(* IEC 61131-3 sources: volt/packages/volt-lsp-iec/test-corpus/lenze-mid/Device/Plc Logic/Application/A70_MachineModuleSources/MM_MachineControl/01_Main, 9 files *)

(* ---- Mach1_Drives.pou ---- *)
FUNCTION_BLOCK Mach1_Drives
VAR_INPUT
END_VAR
VAR_OUTPUT
END_VAR
VAR
	testbyte: BYTE;
	testdint: DWORD;
	testword: WORD;
	OspRotationFlag: R_TRIG;
	OffDelayEnableDrivePower: TOF;
	EnableDrivePower: BOOL;
	bServoDrivesInSync: BOOL;
	TimeOutInSync: TON;
	bInSyncTimeOut: BOOL;
	TimeOutInLock: TON;
	tSetDrivesInLock: BOOL;
	bInLockTimeOut: BOOL;
	SideCorrection_CW: sUDT_ServoComm_Drive_Control;
	Servo_LimitJog_Instance: Servo_LimitJog;
	FBFeedforwardADS: FB_Lenze_i550;
	FBFeedforwardATF: FB_Lenze_i550;
	FBElevatorATF: FB_Lenze_i550;
	FBFan: FB_Lenze_i550;
	FBBobbin: FB_Lenze_i550;
	tReal: REAL;
	tWrapperStopPosition: DINT;

	sadad: FB_Lenze_i550;
	FB_Lenze_i550_0: FB_Lenze_i550;

mydword:DWORD;

	tbool: BOOL;
	OnDelayEnableSync: TON;
	ScaleBobbinTorque: LIN_TRAFO;
	tBobbinTorque: REAL;
	OffDelaySync: TOF;
	TON_0: TON;

	MainDrive_VirtualMasterControl: VirtualMasterControl;
END_VAR

VAR CONSTANT
	ctCurveIsSpeed: INT := 2;
	ctCurveIs0ToMax: INT := 0;
END_VAR
VAR
	ServoMainDrive: ServoControl;
	ServoWrappingDevice: ServoControl;
	ServoSideCorrection: ServoControl;
END_VAR
%LANGUAGE LD
%NETWORK "DONE network 3 : All drives ready"
ASSIGN((Mach1_Data.Drives.MainDrive.Status.DriveIsReady OR INVERT(Mach1_Data.Drives.MainDrive.Control.SetDriveEnable)) AND (Mach1_Data.Drives.WrappingDevice.Status.DriveIsReady OR INVERT(Mach1_Data.Drives.WrappingDevice.Control.SetDriveEnable)) AND (Mach1_Data.Drives.SideCorrection.Status.DriveIsReady OR INVERT(Mach1_Data.Drives.SideCorrection.Control.SetDriveEnable)), Q => Mach1.GenFlags.ConditionsReadyForOperation);
%NETWORK
VAR w1 : ANY; END_VAR
w1 := EnableDrivePower;
ASSIGN(w1 AND Mach1_Data.Drives.WrappingDevice.Status.DriveIsHomed, Q_RESET => Mach1_Data.Drives.WrappingDevice.Control.StartSetHomePos);
ASSIGN((w1 AND INVERT(Mach1_Data.Drives.WrappingDevice.Status.DriveIsHomed)) AND FF500ms, Q_SET => Mach1_Data.Drives.WrappingDevice.Control.StartSetHomePos);
%NETWORK "DONE Network 4: Enable drive power "
// The off delay ensures that the drive can stop before the power is removed from the drive. The power must be removed from the drive before it goes to STO. If the power remains on during STO, the drive will generate an error.
ASSIGN(TRUE AND Mach1_Safety.Status.STO_OK, Q => EnableDrivePower);
%NETWORK
ASSIGN(Mach1_Data.Drives.MainDrive.Status.DriveIsHomed, Q => Mach1_AuxData.AllDrivesHomed);
%NETWORK
VAR w2 : ANY; END_VAR
w2 := TRUE;
ASSIGN(w2 AND mach1.Genflags.DelayAfterSTO, Q => Mach1_Data.Drives.MainDrive_VM.Control.SetDriveEnable);
ASSIGN((w2 AND INVERT(Mach1_Data.Drives.MainDrive_VM.Status.DriveIsReady)) AND FF100ms, Q => Mach1_Data.Drives.MainDrive_VM.Control.ResetError);
MainDrive_VirtualMasterControl(EN := w2, iAcc := 600, iDec := 1800, ioVirtualMaster := Mach1_Data.Drives.MainDrive_VM, ioVirtualMasterCom := Data_Exchange_Motion.Servo_VirtualMaster);
MOVE(EN := MOVE(EN := w2, Mach1_Data.Drives.MainDrive_VM.Status.ActSpeed, OUT => HMI_Var.Mach1.ActualSpeed), Mach1_Data.Drives.MainDrive_VM.Status.ActXPos, OUT => HMI_Var.Mach1.Position);
%NETWORK "Warning: machine in manual homing mode"
Alarms_V5_1_100(AlarmDB := Mach1_Alarms, iCond := Mach1.GenFlags.DelayAfterSTO AND Mach1_AuxData.EnableManualHomeSetting, iReset := Mach1.GenFlags.ResetFlag, iAlm := Mach1_Alarms.Alm033, ioAction := Mach1.GenFlags.Warning);
%NETWORK "DONE Network 5 : Conditions for sync/lock"
VAR w3 : ANY; w4 : ANY; w5 : ANY; END_VAR
w3 := Mach1.GenFlags.DelayAfterEmergStop;
ASSIGN(TON_0(IN := OffDelaySync(IN := w3 AND Mach1_Safety.Status.DoorsOK, PT := T#500MS) AND Mach1_Safety.Status.STO_OK, PT := T#500MS) AND Mach1.GenFlags.ConditionsReadyForOperation AND Mach1_AuxData.AllDrivesHomed AND INVERT(Mach1_AuxData.EnableManualHomeSetting), Q => Mach1_AuxData.SetDrivesInSync);
w4 := w3 AND Mach1_AuxData.SetDrivesInSync;
ASSIGN(w4 AND Mach1_Data.Drives.MainDrive.Status.InSync AND (Mach1_Data.Drives.WrappingDevice.Status.InSync OR INVERT(Mach1_Data.Drives.WrappingDevice.Control.SetDriveEnable)) AND (Mach1_Data.Drives.SideCorrection.Status.InSync OR INVERT(Mach1_Data.Drives.SideCorrection.Control.SetDriveEnable)), Q => bServoDrivesInSync);
ASSIGN(TimeOutInSync(IN := w4 AND INVERT(bServoDrivesInSync), PT := T#10S), Q => bInSyncTimeOut);
ASSIGN(BRANCH_SHORTCIRCUIT(FEED := w3 AND bServoDrivesInSync, Mach1_AuxData.IEC_TIMERS.OffDelayLockDrives(IN := RAIL(), PT := T#2s), TRUE), Q => Mach1_AuxData.SetDrivesInLock);
w5 := w3 AND (Mach1_AuxData.SetDrivesInLock OR Mach1_AuxData.SetDrivesInSync);
ASSIGN(w5 AND Mach1_Data.Drives.MainDrive.Status.InSync AND (Mach1_Data.Drives.WrappingDevice.Status.InSync OR INVERT(Mach1_Data.Drives.WrappingDevice.Control.SetDriveEnable)) AND (Mach1_Data.Drives.SideCorrection.Status.InSync OR INVERT(Mach1_Data.Drives.SideCorrection.Control.SetDriveEnable)), Q => Mach1_AuxData.AllDrivesInLock);
ASSIGN(TimeOutInLock(IN := w5 AND INVERT(Mach1_AuxData.AllDrivesInLock), PT := T#5S), Q => bInLockTimeOut);
ASSIGN(w5, Q => tSetDrivesInLock);
%NETWORK "DONE Network 6: Servo Main drive: Control"
VAR w6 : ANY; w7 : ANY; END_VAR
w6 := TRUE;
ASSIGN(w6 AND (Mach1_Safety.Control.RequestManSpeed AND Mach1_Safety.Status.SafetyManSpeed OR Mach1_Safety.Control.RequestAutoSpeed AND Mach1_Safety.Status.SafetyAutoSpeed), Q => Mach1_Data.Drives.MainDrive_VM.Control.StartMovement);
ASSIGN(MOVE(EN := w6 AND TRUE, ctCurveIs0ToMax, OUT => Mach1_Data.Drives.MainDrive.CAM.CamType) AND tSetDrivesInLock, Q => Mach1_Data.Drives.MainDrive.Control.SetInSync);
w7 := w6 AND TRUE;
ASSIGN(w7 AND Mach1_Alarms.Alm001 AND HMI_Var.ReleaseBrake, Q => Mach1_Data.Drives.MainDrive.Control.SetBrakeRelease);
ASSIGN(w7 AND (INVERT(Mach1_Alarms.Alm001) OR mach1.Genflags.StartFlag AND Mach1_Alarms.Alm001), Q_RESET => HMI_Var.ReleaseBrake);
ASSIGN(OspRotationFlag(CLK := ServoMainDrive(EN := w6 AND TRUE, iServoStatus := Data_Exchange_Motion.Servo_MainDrive.Status, iEnableHomeMovement := TRUE, iEnablePower := EnableDrivePower, iFF100ms := LST_General.FF100ms, ioUDT_ServoDrive := Mach1_Data.Drives.MainDrive, oServoControl => Data_Exchange_Motion.Servo_MainDrive.Control) AND Mach1_Data.Drives.MainDrive.Status.RotationPulse), Q => Mach1.GenFlags.Rotflag);
%NETWORK "DONE Network 7 : Servo Main drive: Alarms"
ASSIGN(Alarms_V5_1_100(AlarmDB := Mach1_Alarms, iCond := Mach1.GenFlags.DelayAfterSTO AND INVERT(Mach1_Data.Drives.MainDrive.Status.DriveIsReady), iReset := Mach1.GenFlags.ResetFlag, iAlm := Mach1_Alarms.Alm020, ioAction := Mach1.GenFlags.MinorAlarm) OR Alarms_V5_1_100(AlarmDB := Mach1_Alarms, iCond := Mach1.GenFlags.DelayAfterSTO AND Mach1_Data.Drives.MainDrive.Status.DriveTorqueError, iReset := Mach1.GenFlags.ResetFlag, iAlm := Mach1_Alarms.Alm021, ioAction := Mach1.GenFlags.MinorAlarm) OR Alarms_V5_1_100(AlarmDB := Mach1_Alarms, iCond := Mach1.GenFlags.DelayAfterSTO AND INVERT(Mach1_Data.Drives.MainDrive.Status.DriveIsHomed), iReset := Mach1.GenFlags.ResetFlag, iAlm := Mach1_Alarms.Alm022, ioAction := Mach1.GenFlags.MinorAlarm), Q_SET => Mach1.GenFlags.StopDriveDirect);
%NETWORK
ASSIGN((Mach1_Alarms.Alm020 OR Mach1_Alarms.Alm021 OR Mach1_Alarms.Alm022) AND Mach1.GenFlags.ResetFlag OR TON_0.Q AND Imp100ms AND Mach1_Safety.Status.ServiceMode AND Mach1_Safety.Status.Service_ButtonAB, Q_SET => Mach1_Data.Drives.MainDrive.Control.ResetError);
%NETWORK "DONE Network 8: Servo Wrapping device: Control"
VAR w8 : ANY; END_VAR
w8 := TRUE;
ASSIGN(MOVE(EN := w8 AND TRUE, ctCurveIsSpeed, OUT => Mach1_Data.Drives.WrappingDevice.CAM.CamType) AND tSetDrivesInLock, Q => Mach1_Data.Drives.WrappingDevice.Control.SetInSync);
MOVE(EN := w8, Mach1_Data.Settings.Ints.RollingDeviceSpeedFactor, OUT => Mach1_Data.Drives.WrappingDevice.CAM.Y_Scale_Recipe);
ServoWrappingDevice(EN := w8 AND TRUE, iServoStatus := Data_Exchange_Motion.Servo_WrappingDevice.Status, iEnableHomeMovement := TRUE, iEnablePower := EnableDrivePower, iFF100ms := LST_General.FF100ms, ioUDT_ServoDrive := Mach1_Data.Drives.WrappingDevice, oServoControl => Data_Exchange_Motion.Servo_WrappingDevice.Control);
%NETWORK "DONE Network 9 : Servo Wrapping Device: Alarms"
VAR w9 : ANY; END_VAR
w9 := Alarms_V5_1_100(AlarmDB := Mach1_Alarms, iCond := Mach1.GenFlags.DelayAfterSTO AND INVERT(Mach1_Data.Drives.WrappingDevice.Status.DriveIsReady) AND Mach1_Data.Drives.WrappingDevice.Control.SetDriveEnable, iReset := Mach1.GenFlags.ResetFlag, iAlm := Mach1_Alarms.Alm023, ioAction := Mach1.GenFlags.MinorAlarm) OR Alarms_V5_1_100(AlarmDB := Mach1_Alarms, iCond := Mach1.GenFlags.DelayAfterSTO AND Mach1_Data.Drives.WrappingDevice.Status.DriveTorqueError, iReset := Mach1.GenFlags.ResetFlag, iAlm := Mach1_Alarms.Alm024, ioAction := Mach1.GenFlags.MinorAlarm) OR Alarms_V5_1_100(AlarmDB := Mach1_Alarms, iCond := Mach1.GenFlags.DelayAfterSTO AND INVERT(Mach1_Data.Drives.WrappingDevice.Status.DriveIsHomed), iReset := Mach1.GenFlags.ResetFlag, iAlm := Mach1_Alarms.Alm025, ioAction := Mach1.GenFlags.MinorAlarm);
ASSIGN(w9, Q_SET => Mach1.GenFlags.StopDriveDirect);
ASSIGN(w9 AND Mach1.GenFlags.ResetFlag, Q_SET => Mach1_Data.Drives.WrappingDevice.Control.ResetError);
%NETWORK
ASSIGN((Mach1_Alarms.Alm023 OR Mach1_Alarms.Alm024 OR Mach1_Alarms.Alm025) AND Mach1.GenFlags.ResetFlag OR TON_0.Q AND Imp100ms AND Mach1_Safety.Status.ServiceMode AND Mach1_Safety.Status.Service_ButtonAB, Q_SET => Mach1_Data.Drives.WrappingDevice.Control.ResetError);
%NETWORK
%NETWORK "Digital inputs"
VAR w10 : ANY; END_VAR
// 16: non-motor side
// 17: motor side
w10 := MOVE(EN := TRUE, %ID79, OUT => mydword);
ASSIGN(w10 AND mydword.16, Q => Data_Exchange_Motion.Servo_SideCorrection.Status.Spare1);
ASSIGN(w10 AND mydword.17, Q => Data_Exchange_Motion.Servo_SideCorrection.Status.Spare2);
%NETWORK "DONE Network 10: Servo Side correction: Control"
VAR w11 : ANY; END_VAR
w11 := TRUE;
ASSIGN(MOVE(EN := w11 AND TRUE, ctCurveIsSpeed, OUT => Mach1_Data.Drives.SideCorrection.CAM.CamType) AND tSetDrivesInLock, Q => Mach1_Data.Drives.SideCorrection.Control.SetInSync);
ServoSideCorrection(EN := w11 AND TRUE, iServoStatus := Data_Exchange_Motion.Servo_SideCorrection.Status, iEnableHomeMovement := TRUE, iEnablePower := EnableDrivePower, iFF100ms := LST_General.FF100ms, ioUDT_ServoDrive := Mach1_Data.Drives.SideCorrection, oServoControl => SideCorrection_CW);
Servo_LimitJog_Instance(EN := w11 AND TRUE, iServoStatus := Data_Exchange_Motion.Servo_SideCorrection.Status, iServoControl := SideCorrection_CW, ioUDT_ServoDrive := Mach1_Data.Drives.SideCorrection, ioUDT_JogLimitFree := Mach1_Data.Drives.SideCorrection_FreeLimit, oServoControl => Data_Exchange_Motion.Servo_SideCorrection.Control);
%NETWORK "DONE Network 11 : Servo Side correction: Alarms"
VAR w12 : ANY; END_VAR
w12 := Alarms_V5_1_100(AlarmDB := Mach1_Alarms, iCond := Mach1.GenFlags.DelayAfterSTO AND INVERT(Mach1_Data.Drives.SideCorrection.Status.DriveIsReady) AND Mach1_Data.Drives.SideCorrection.Control.SetDriveEnable, iReset := Mach1.GenFlags.ResetFlag, iAlm := Mach1_Alarms.Alm026, ioAction := Mach1.GenFlags.MinorAlarm) OR Alarms_V5_1_100(AlarmDB := Mach1_Alarms, iCond := Mach1.GenFlags.DelayAfterSTO AND Mach1_Data.Drives.SideCorrection.Status.DriveTorqueError, iReset := Mach1.GenFlags.ResetFlag, iAlm := Mach1_Alarms.Alm027, ioAction := Mach1.GenFlags.MinorAlarm) OR Alarms_V5_1_100(AlarmDB := Mach1_Alarms, iCond := Mach1.GenFlags.DelayAfterSTO AND INVERT(Mach1_Data.Drives.SideCorrection.Status.DriveIsHomed), iReset := Mach1.GenFlags.ResetFlag, iAlm := Mach1_Alarms.Alm028, ioAction := Mach1.GenFlags.MinorAlarm);
ASSIGN(w12, Q_SET => Mach1.GenFlags.StopDriveDirect);
ASSIGN(w12 AND Mach1.GenFlags.ResetFlag, Q_SET => Mach1_Data.Drives.SideCorrection.Control.ResetError);
%NETWORK
ASSIGN((Mach1_Alarms.Alm026 OR Mach1_Alarms.Alm027 OR Mach1_Alarms.Alm028) AND Mach1.GenFlags.ResetFlag OR TON_0.Q AND Imp100ms AND Mach1_Safety.Status.ServiceMode AND Mach1_Safety.Status.Service_ButtonAB, Q_SET => Mach1_Data.Drives.SideCorrection.Control.ResetError);
%NETWORK
%NETWORK "DONE Network 12: Feedforward ADS"
VAR w13 : ANY; END_VAR
w13 := TRUE;
ASSIGN(w13 AND Mach1.GenFlags.DelayAfterEmergStop AND INVERT(Mach1_Alarms.Alm015), Q => Mach1_Data.Drives.FeedForwardADS.Control.Enable);
ASSIGN(w13, Q => Mach1_Data.Drives.FeedForwardADS.Control.Reverse);
FBFeedforwardADS(EN := w13, iStatusWord := Data_Exchange_Motion.FQI_FeedforwardADS.Status, iGearRatioNumerator := 2790.0, iGearRatioDenominator := 111.0, iNominalMotorSpeedwoSlipComp_RPM := 3000.0, iNominalMotorFrequency_Hz := 100.0, iAxisJogSpeed_RPM := 10.0, ioUDT := Mach1_Data.Drives.FeedForwardADS, oControlWord => Data_Exchange_Motion.FQI_FeedforwardADS.Controlword, oRefSpeed => Data_Exchange_Motion.FQI_FeedforwardADS.RefSpeed);
%NETWORK "DONE Network 13: Alarms feed forward dryer "
VAR w14 : ANY; END_VAR
w14 := Alarms_V5_1_100(AlarmDB := Mach1_Alarms, iCond := Mach1.GenFlags.DelayAfterEmergStop AND Mach1_Data.Drives.FeedForwardADS.Status.Error, iReset := True, iAlm := Mach1_Alarms.Alm015, ioAction := Mach1.GenFlags.MinorAlarm);
ASSIGN(w14, Q_SET => Mach1.GenFlags.StopDriveDirect);
ASSIGN(w14 AND Mach1.GenFlags.ResetFlag, Q_SET => Mach1_Data.Drives.FeedForwardADS.Control.ResetError);
%NETWORK "DONE Network 14: Feedforward ATF"
VAR w15 : ANY; END_VAR
w15 := TRUE;
ASSIGN(w15 AND Mach1.GenFlags.DelayAfterEmergStop AND INVERT(Mach1_Alarms.Alm016), Q => Mach1_Data.Drives.FeedForwardATF.Control.Enable);
FBFeedforwardATF(EN := w15, iStatusWord := Data_Exchange_Motion.FQI_FeedforwardATF.Status, iGearRatioNumerator := 2790.0, iGearRatioDenominator := 111.0, iNominalMotorSpeedwoSlipComp_RPM := 3000.0, iNominalMotorFrequency_Hz := 100.0, iAxisJogSpeed_RPM := 10.0, ioUDT := Mach1_Data.Drives.FeedForwardATF, oControlWord => Data_Exchange_Motion.FQI_FeedforwardATF.Controlword, oRefSpeed => Data_Exchange_Motion.FQI_FeedforwardATF.RefSpeed);
%NETWORK "DONE Network 15: Alarms feed forward trayfiller$R$L"
VAR w16 : ANY; END_VAR
w16 := Alarms_V5_1_100(AlarmDB := Mach1_Alarms, iCond := Mach1.GenFlags.DelayAfterEmergStop AND Mach1_Data.Drives.FeedForwardATF.Status.Error, iReset := True, iAlm := Mach1_Alarms.Alm016, ioAction := Mach1.GenFlags.MinorAlarm);
ASSIGN(w16, Q_SET => Mach1.GenFlags.StopDriveDirect);
ASSIGN(w16 AND Mach1.GenFlags.ResetFlag, Q_SET => Mach1_Data.Drives.FeedForwardATF.Control.ResetError);
%NETWORK "DONE Network 16: Elevator ATF"
VAR w17 : ANY; END_VAR
w17 := TRUE;
ASSIGN(w17 AND Mach1.GenFlags.DelayAfterEmergStop AND INVERT(Mach1_Alarms.Alm014), Q => Mach1_Data.Drives.ElevatorATF.Control.Enable);
FBElevatorATF(EN := w17, iStatusWord := Data_Exchange_Motion.FQI_ElevatorATF.Status, iGearRatioNumerator := 100.0, iGearRatioDenominator := 111.0, iNominalMotorSpeedwoSlipComp_RPM := 3000.0, iNominalMotorFrequency_Hz := 100.0, iAxisJogSpeed_RPM := 10.0, ioUDT := Mach1_Data.Drives.ElevatorATF, oControlWord => Data_Exchange_Motion.FQI_ElevatorATF.Controlword, oRefSpeed => Data_Exchange_Motion.FQI_ElevatorATF.RefSpeed);
%NETWORK "DONE Network 17: Alarms Elevator trayfiller$R$L"
VAR w18 : ANY; END_VAR
w18 := Alarms_V5_1_100(AlarmDB := Mach1_Alarms, iCond := Mach1.GenFlags.DelayAfterEmergStop AND Mach1_Data.Drives.ElevatorATF.Status.Error, iReset := True, iAlm := Mach1_Alarms.Alm014, ioAction := Mach1.GenFlags.MinorAlarm);
ASSIGN(w18, Q_SET => Mach1.GenFlags.StopDriveDirect);
ASSIGN(w18 AND Mach1.GenFlags.ResetFlag, Q_SET => Mach1_Data.Drives.ElevatorATF.Control.ResetError);
%NETWORK "DONE Network 18: Fan"
VAR w19 : ANY; END_VAR
w19 := TRUE;
ASSIGN(w19 AND Mach1.GenFlags.EnableAuxDrive AND INVERT(Mach1_Alarms.Alm017), Q => Mach1_Data.Drives.Fan.Control.Enable);
FBFan(EN := w19, iStatusWord := Data_Exchange_Motion.FQI_Fan.Status, iGearRatioNumerator := 1.0, iGearRatioDenominator := 1.0, iNominalMotorSpeedwoSlipComp_RPM := 3000.0, iNominalMotorFrequency_Hz := 50.0, iAxisJogSpeed_RPM := 10.0, ioUDT := Mach1_Data.Drives.Fan, oControlWord => Data_Exchange_Motion.FQI_Fan.Controlword, oRefSpeed => Data_Exchange_Motion.FQI_Fan.RefSpeed);
%NETWORK "DONE Network 19: Alarms Fan$R$L"
VAR w20 : ANY; END_VAR
w20 := Alarms_V5_1_100(AlarmDB := Mach1_Alarms, iCond := Mach1.GenFlags.DelayAfterEmergStop AND Mach1_Data.Drives.Fan.Status.Error, iReset := True, iAlm := Mach1_Alarms.Alm017, ioAction := Mach1.GenFlags.MinorAlarm);
ASSIGN(w20, Q_SET => Mach1.GenFlags.StopDriveDirect);
ASSIGN(w20 AND Mach1.GenFlags.ResetFlag, Q_SET => Mach1_Data.Drives.Fan.Control.ResetError);
%NETWORK "DONE Network 20: Bobbin"
VAR w21 : ANY; w22 : ANY; w23 : ANY; END_VAR
w21 := TRUE;
w22 := GT(EN := w21 AND Mach1.GenFlags.EnableAuxDrive AND INVERT(HMI_Var.Btn_Cleaning), Mach1_Data.Settings.Ints.TorqueControlBobbin, 0).OUT AND Mach1_Safety.Status.AllDoorsActuallyClosed;
ASSIGN(w22, Q => Mach1_Data.Drives.Bobbine.Control.Enable);
ASSIGN(MOVE(EN := w22, 860, OUT => Mach1_Data.Drives.Bobbine.Control.AutoSpeed), Q => Mach1_Data.Drives.Bobbine.Control.StartAuto);
FBBobbin(EN := w21, iStatusWord := Data_Exchange_Motion.FQI_Bobbin.Status, iGearRatioNumerator := 2790.0, iGearRatioDenominator := 111.0, iNominalMotorSpeedwoSlipComp_RPM := 3000.0, iNominalMotorFrequency_Hz := 50.0, iAxisJogSpeed_RPM := 10.0, ioUDT := Mach1_Data.Drives.Bobbine, oControlWord => Data_Exchange_Motion.FQI_Bobbin.Controlword, oRefSpeed => Data_Exchange_Motion.FQI_Bobbin.RefSpeed);
w23 := w21 AND HMI_Var.Mach1.CalibrateTorqueValues;
MOVE(EN := w23, Mach1_AuxData.TorqueCalibrationValue, OUT => Data_Exchange_Motion.BobbinTorque);
ASSIGN(MOVE(EN := w23 AND HMI_Var.Mach1.setMinTorqueValue, Mach1_AuxData.TorqueCalibrationValue, OUT => Mach1_Data.Settings.Dints.minTorqueValue), Q_RESET => HMI_Var.Mach1.setMinTorqueValue);
ASSIGN(MOVE(EN := w23 AND HMI_Var.Mach1.setMaxTorqueValue, Mach1_AuxData.TorqueCalibrationValue, OUT => Mach1_Data.Settings.Dints.maxTorqueValue), Q_RESET => HMI_Var.Mach1.setMaxTorqueValue);
MOVE(EN := ScaleBobbinTorque(EN := w21 AND INVERT(HMI_Var.Mach1.CalibrateTorqueValues), IN := Mach1_Data.Settings.Ints.TorqueControlBobbin, IN_MIN := 0, IN_MAX := 1000, OUT_MIN := OPERAND('DINT_TO_REAL(Mach1_Data.Settings.Dints.minTorqueValue)'), OUT_MAX := OPERAND('DINT_TO_REAL(Mach1_Data.Settings.Dints.maxTorqueValue)'), OUT => tBobbinTorque), OPERAND('REAL_TO_DINT(tBobbinTorque)'), OUT => Data_Exchange_Motion.BobbinTorque);
%NETWORK "DONE Network 21: Alarms Bobbine $R$L"
VAR w24 : ANY; END_VAR
w24 := Alarms_V5_1_100(AlarmDB := Mach1_Alarms, iCond := Mach1_AuxData.MIDS_Active AND Mach1.GenFlags.DelayAfterEmergStop AND INVERT(Mach1_Data.Drives.Bobbine.Status.DriveReady) AND Mach1_AuxData.AllDrivesHomed, iReset := True, iAlm := Mach1_Alarms.Alm010, ioAction := Mach1.GenFlags.MinorAlarm);
ASSIGN(w24, Q_SET => Mach1.GenFlags.StopDriveDirect);
ASSIGN(w24 AND Mach1.GenFlags.ResetFlag, Q_SET => Mach1_Data.Drives.Bobbine.Control.ResetError);
%NETWORK "TODO Network 22:"
// WRAPPER
%NETWORK "TODO Network 23: Limit Wrapper stop position"
VAR w25 : ANY; END_VAR
w25 := TRUE;
MOVE(EN := GT(EN := w25, Mach1_Data.Settings.Dints.WrapperStopPosition, 400).OUT, 400, OUT => Mach1_Data.Settings.Dints.WrapperStopPosition);
MOVE(EN := LT(EN := w25, Mach1_Data.Settings.Dints.WrapperStopPosition, 5).OUT, 5, OUT => Mach1_Data.Settings.Dints.WrapperStopPosition);
MUL(EN := w25, Mach1_Data.Settings.Dints.WrapperStopPosition, 100, OUT => tWrapperStopPosition);
%NETWORK "TODO Network 25:"
ASSIGN(TRUE AND Mach1.GenFlags.DelayAfterEmergStop AND INVERT(Mach1_Alarms.Alm066), Q => Data_Exchange_Motion.FeedForwardWrapper.Control.Enable);
%NETWORK "TODO Network 26:"
ASSIGN(Alarms_V5_1_100(AlarmDB := Mach1_Alarms, iCond := Mach1_AuxData.MIDS_Active AND Mach1.GenFlags.EnableMainDrive AND HMI_Var.Test_Prod AND INVERT(HMI_Var.Btn_Cleaning) AND Mach1_AuxData.AllDrivesHomed AND INVERT(Data_Exchange_Motion.FeedForwardWrapper.Status.ReadyForMotion), iReset := Mach1.Genflags.StartFlag, iAlm := Mach1_Alarms.Alm056, ioAction := Mach1.GenFlags.MinorAlarm) AND mach1.Genflags.ResetFlag, Q_SET => Mach1_Data.Drives.WrappingDevice.Control.ResetError, Q => Data_Exchange_Motion.FeedForwardWrapper.Control.ResetError);
%NETWORK "TODO Network 27:"
;

END_FUNCTION_BLOCK

(* ---- fc_Information.pou ---- *)
PROGRAM fc_Information
VAR
END_VAR

%LANGUAGE ST
VersionInfo_DB.PLC_version:='MID-S100-L-V00_00';
VersionInfo_DB.PLC_Version_Date:='08-06-2023';

END_PROGRAM

(* ---- ForceOutput.pou ---- *)
PROGRAM ForceOutput
VAR
END_VAR

%LANGUAGE LD
%NETWORK
VAR w1 : ANY; END_VAR
w1 := HMI_Var.ForceOutputs;
ASSIGN(w1 AND LST_InputsOutputs.Serv_QB100.0, Q => LST_InputsOutputs.Q100_0_Pilot_light_Alarm_green_);
ASSIGN(w1 AND LST_InputsOutputs.Serv_QB100.1, Q => LST_InputsOutputs.Q100_1_Pilot_light_Alarm_orange_);
ASSIGN(w1 AND LST_InputsOutputs.Serv_QB100.2, Q => LST_InputsOutputs.Q100_2_Pilot_light_Alarm_red_);
ASSIGN(w1 AND LST_InputsOutputs.Serv_QB100.3, Q => LST_InputsOutputs.Q100_3_Pilot_light_Alarm_buzzer_);
ASSIGN(w1 AND LST_InputsOutputs.Serv_QB100.4, Q => LST_InputsOutputs.Q100_4_Spare);
ASSIGN(w1 AND LST_InputsOutputs.Serv_QB100.5, Q => LST_InputsOutputs.Q100_5_Signal_lamp_Start);
ASSIGN(w1 AND LST_InputsOutputs.Serv_QB100.6, Q => LST_InputsOutputs.Q100_6_Signal_lamp_Stop);
ASSIGN(w1 AND LST_InputsOutputs.Serv_QB100.7, Q => LST_InputsOutputs.Q100_7_Activate_greasing_system);
ASSIGN(w1 AND LST_InputsOutputs.Serv_QB101.0, Q => LST_InputsOutputs.Q101_0_REL_release_brake);
ASSIGN(w1 AND LST_InputsOutputs.Serv_QB101.1, Q => LST_InputsOutputs.Q101_1_PNV_Waterlevel_control);
ASSIGN(w1 AND LST_InputsOutputs.Serv_QB101.2, Q => LST_InputsOutputs.Q101_2_Enable_GluePump);
ASSIGN(w1 AND LST_InputsOutputs.Serv_QB101.3, Q => LST_InputsOutputs.Q101_3_Spare);
ASSIGN(w1 AND LST_InputsOutputs.Serv_QB101.4, Q => LST_InputsOutputs.Q101_4_Spare);
ASSIGN(w1 AND LST_InputsOutputs.Serv_QB101.5, Q => LST_InputsOutputs.Q101_5_Spare);
ASSIGN(w1 AND LST_InputsOutputs.Serv_QB101.6, Q => LST_InputsOutputs.Q101_6_Spare);
ASSIGN(w1 AND LST_InputsOutputs.Serv_QB101.7, Q => LST_InputsOutputs.Q101_7_Spare);
%NETWORK
VAR w2 : ANY; END_VAR
w2 := HMI_Var.ForceOutputs;
ASSIGN(w2 AND LST_InputsOutputs.Serv_QB132.0, Q => LST_InputsOutputs.Q132_0_SL_Start_OP2a);
ASSIGN(w2 AND LST_InputsOutputs.Serv_QB132.1, Q => LST_InputsOutputs.Q132_1_SL_Stop_OP2a);
ASSIGN(w2 AND LST_InputsOutputs.Serv_QB132.2, Q => LST_InputsOutputs.Q132_2_Enable_power_controllers);
ASSIGN(w2 AND LST_InputsOutputs.Serv_QB132.3, Q => LST_InputsOutputs.Q132_3_Spare);
ASSIGN(w2 AND LST_InputsOutputs.Serv_QB132.4, Q => LST_InputsOutputs.Q132_4_CT_Fan_dryer);
ASSIGN(w2 AND LST_InputsOutputs.Serv_QB132.5, Q => LST_InputsOutputs.Q132_5_Spare);
ASSIGN(w2 AND LST_InputsOutputs.Serv_QB132.6, Q => LST_InputsOutputs.Q132_6_PNV_Inpusher);
ASSIGN(w2 AND LST_InputsOutputs.Serv_QB132.7, Q => LST_InputsOutputs.Q132_7_PNV_tilting_inpusher);
ASSIGN(w2 AND LST_InputsOutputs.Serv_QB133.0, Q => LST_InputsOutputs.Q133_0_Spare);
ASSIGN(w2 AND LST_InputsOutputs.Serv_QB133.1, Q => LST_InputsOutputs.Q133_1_Spare);
ASSIGN(w2 AND LST_InputsOutputs.Serv_QB133.2, Q => LST_InputsOutputs.Q133_2_Spare);
ASSIGN(w2 AND LST_InputsOutputs.Serv_QB133.3, Q => LST_InputsOutputs.Q133_3_Spare);
ASSIGN(w2 AND LST_InputsOutputs.Serv_QB133.4, Q => LST_InputsOutputs.Q133_4_Spare);
ASSIGN(w2 AND LST_InputsOutputs.Serv_QB133.5, Q => LST_InputsOutputs.Q133_5_InfeedConv_Fwd);
ASSIGN(w2 AND LST_InputsOutputs.Serv_QB133.6, Q => LST_InputsOutputs.Q133_6_InfeedConv_Rev);
ASSIGN(w2 AND LST_InputsOutputs.Serv_QB133.7, Q => LST_InputsOutputs.Q133_7_OutfeedConv_Fwd);
%NETWORK
VAR w3 : ANY; END_VAR
w3 := HMI_Var.ForceOutputs;
ASSIGN(w3 AND LST_InputsOutputs.Serv_QB136.0, Q => LST_InputsOutputs.Q136_0_Spare);
ASSIGN(w3 AND LST_InputsOutputs.Serv_QB136.1, Q => LST_InputsOutputs.Q136_1_Spare);
ASSIGN(w3 AND LST_InputsOutputs.Serv_QB136.2, Q => LST_InputsOutputs.Q136_2_Spare);
ASSIGN(w3 AND LST_InputsOutputs.Serv_QB136.3, Q => LST_InputsOutputs.Q136_3_Spare);
ASSIGN(w3 AND LST_InputsOutputs.Serv_QB136.4, Q => LST_InputsOutputs.Q136_4_Spare);
ASSIGN(w3 AND LST_InputsOutputs.Serv_QB136.5, Q => LST_InputsOutputs.Q136_5_Spare);
ASSIGN(w3 AND LST_InputsOutputs.Serv_QB136.6, Q => LST_InputsOutputs.Q136_6_Spare);
ASSIGN(w3 AND LST_InputsOutputs.Serv_QB132.7, Q => LST_InputsOutputs.Q136_7_Spare);
ASSIGN(w3 AND LST_InputsOutputs.Serv_QB137.0, Q => LST_InputsOutputs.Q137_0_Spare);
ASSIGN(w3 AND LST_InputsOutputs.Serv_QB137.1, Q => LST_InputsOutputs.Q137_1_Spare);
ASSIGN(w3 AND LST_InputsOutputs.Serv_QB137.2, Q => LST_InputsOutputs.Q137_2_Spare);
ASSIGN(w3 AND LST_InputsOutputs.Serv_QB137.3, Q => LST_InputsOutputs.Q137_3_Spare);
ASSIGN(w3 AND LST_InputsOutputs.Serv_QB137.4, Q => LST_InputsOutputs.Q137_4_Spare);
ASSIGN(w3 AND LST_InputsOutputs.Serv_QB137.5, Q => LST_InputsOutputs.Q137_5_Spare);
ASSIGN(w3 AND LST_InputsOutputs.Serv_QB137.6, Q => LST_InputsOutputs.Q137_6_Spare);
ASSIGN(w3 AND LST_InputsOutputs.Serv_QB137.7, Q => LST_InputsOutputs.Q137_7_Spare);
%NETWORK

END_PROGRAM

(* ---- ForceOutput_1.pou ---- *)
PROGRAM ForceOutput_1
VAR
END_VAR

%LANGUAGE LD
%NETWORK
VAR w1 : ANY; END_VAR
w1 := INVERT(HMI_Var.ForceOutputs);
ASSIGN(w1 AND LST_InputsOutputs.Q100_0_Pilot_light_Alarm_green_, Q => LST_InputsOutputs.Serv_QB100.0);
ASSIGN(w1 AND LST_InputsOutputs.Q100_1_Pilot_light_Alarm_orange_, Q => LST_InputsOutputs.Serv_QB100.1);
ASSIGN(w1 AND LST_InputsOutputs.Q100_2_Pilot_light_Alarm_red_, Q => LST_InputsOutputs.Serv_QB100.2);
ASSIGN(w1 AND LST_InputsOutputs.Q100_3_Pilot_light_Alarm_buzzer_, Q => LST_InputsOutputs.Serv_QB100.3);
ASSIGN(w1 AND LST_InputsOutputs.Q100_4_Spare, Q => LST_InputsOutputs.Serv_QB100.4);
ASSIGN(w1 AND LST_InputsOutputs.Q100_5_Signal_lamp_Start, Q => LST_InputsOutputs.Serv_QB100.5);
ASSIGN(w1 AND LST_InputsOutputs.Q100_6_Signal_lamp_Stop, Q => LST_InputsOutputs.Serv_QB100.6);
ASSIGN(w1 AND LST_InputsOutputs.Q100_7_Activate_greasing_system, Q => LST_InputsOutputs.Serv_QB100.7);
ASSIGN(w1 AND LST_InputsOutputs.Q101_0_REL_release_brake, Q => LST_InputsOutputs.Serv_QB101.0);
ASSIGN(w1 AND LST_InputsOutputs.Q101_1_PNV_Waterlevel_control, Q => LST_InputsOutputs.Serv_QB101.1);
ASSIGN(w1 AND LST_InputsOutputs.Q101_2_Enable_GluePump, Q => LST_InputsOutputs.Serv_QB101.2);
ASSIGN(w1 AND LST_InputsOutputs.Q101_3_Spare, Q => LST_InputsOutputs.Serv_QB101.3);
ASSIGN(w1 AND LST_InputsOutputs.Q101_4_Spare, Q => LST_InputsOutputs.Serv_QB101.4);
ASSIGN(w1 AND LST_InputsOutputs.Q101_5_Spare, Q => LST_InputsOutputs.Serv_QB101.5);
ASSIGN(w1 AND LST_InputsOutputs.Q101_6_Spare, Q => LST_InputsOutputs.Serv_QB101.6);
ASSIGN(w1 AND LST_InputsOutputs.Q101_7_Spare, Q => LST_InputsOutputs.Serv_QB101.7);
%NETWORK
VAR w2 : ANY; END_VAR
w2 := INVERT(HMI_Var.ForceOutputs);
ASSIGN(w2 AND LST_InputsOutputs.Q132_0_SL_Start_OP2a, Q => LST_InputsOutputs.Serv_QB132.0);
ASSIGN(w2 AND LST_InputsOutputs.Q132_1_SL_Stop_OP2a, Q => LST_InputsOutputs.Serv_QB132.1);
ASSIGN(w2 AND LST_InputsOutputs.Q132_2_Enable_power_controllers, Q => LST_InputsOutputs.Serv_QB132.2);
ASSIGN(w2 AND LST_InputsOutputs.Q132_3_Spare, Q => LST_InputsOutputs.Serv_QB132.3);
ASSIGN(w2 AND LST_InputsOutputs.Q132_4_CT_Fan_dryer, Q => LST_InputsOutputs.Serv_QB132.4);
ASSIGN(w2 AND LST_InputsOutputs.Q132_5_Spare, Q => LST_InputsOutputs.Serv_QB132.5);
ASSIGN(w2 AND LST_InputsOutputs.Q132_6_PNV_Inpusher, Q => LST_InputsOutputs.Serv_QB132.6);
ASSIGN(w2 AND LST_InputsOutputs.Q132_7_PNV_tilting_inpusher, Q => LST_InputsOutputs.Serv_QB132.7);
ASSIGN(w2 AND LST_InputsOutputs.Q133_0_Spare, Q => LST_InputsOutputs.Serv_QB133.0);
ASSIGN(w2 AND LST_InputsOutputs.Q133_1_Spare, Q => LST_InputsOutputs.Serv_QB133.1);
ASSIGN(w2 AND LST_InputsOutputs.Q133_2_Spare, Q => LST_InputsOutputs.Serv_QB133.2);
ASSIGN(w2 AND LST_InputsOutputs.Q133_3_Spare, Q => LST_InputsOutputs.Serv_QB133.3);
ASSIGN(w2 AND LST_InputsOutputs.Q133_4_Spare, Q => LST_InputsOutputs.Serv_QB133.4);
ASSIGN(w2 AND LST_InputsOutputs.Q133_5_InfeedConv_Fwd, Q => LST_InputsOutputs.Serv_QB133.5);
ASSIGN(w2 AND LST_InputsOutputs.Q133_6_InfeedConv_Rev, Q => LST_InputsOutputs.Serv_QB133.6);
ASSIGN(w2 AND LST_InputsOutputs.Q133_7_OutfeedConv_Fwd, Q => LST_InputsOutputs.Serv_QB133.7);
%NETWORK
VAR w3 : ANY; END_VAR
w3 := INVERT(HMI_Var.ForceOutputs);
ASSIGN(w3 AND LST_InputsOutputs.Q136_0_Spare, Q => LST_InputsOutputs.Serv_QB136.0);
ASSIGN(w3 AND LST_InputsOutputs.Q136_1_Spare, Q => LST_InputsOutputs.Serv_QB136.1);
ASSIGN(w3 AND LST_InputsOutputs.Q136_2_Spare, Q => LST_InputsOutputs.Serv_QB136.2);
ASSIGN(w3 AND LST_InputsOutputs.Q136_3_Spare, Q => LST_InputsOutputs.Serv_QB136.3);
ASSIGN(w3 AND LST_InputsOutputs.Q136_4_Spare, Q => LST_InputsOutputs.Serv_QB136.4);
ASSIGN(w3 AND LST_InputsOutputs.Q136_5_Spare, Q => LST_InputsOutputs.Serv_QB136.5);
ASSIGN(w3 AND LST_InputsOutputs.Q136_6_Spare, Q => LST_InputsOutputs.Serv_QB136.6);
ASSIGN(w3 AND LST_InputsOutputs.Q136_7_Spare, Q => LST_InputsOutputs.Serv_QB132.7);
ASSIGN(w3 AND LST_InputsOutputs.Q137_0_Spare, Q => LST_InputsOutputs.Serv_QB137.0);
ASSIGN(w3 AND LST_InputsOutputs.Q137_1_Spare, Q => LST_InputsOutputs.Serv_QB137.1);
ASSIGN(w3 AND LST_InputsOutputs.Q137_2_Spare, Q => LST_InputsOutputs.Serv_QB137.2);
ASSIGN(w3 AND LST_InputsOutputs.Q137_3_Spare, Q => LST_InputsOutputs.Serv_QB137.3);
ASSIGN(w3 AND LST_InputsOutputs.Q137_4_Spare, Q => LST_InputsOutputs.Serv_QB137.4);
ASSIGN(w3 AND LST_InputsOutputs.Q137_5_Spare, Q => LST_InputsOutputs.Serv_QB137.5);
ASSIGN(w3 AND LST_InputsOutputs.Q137_6_Spare, Q => LST_InputsOutputs.Serv_QB137.6);
ASSIGN(w3 AND LST_InputsOutputs.Q137_7_Spare, Q => LST_InputsOutputs.Serv_QB137.7);
%NETWORK

END_PROGRAM

(* ---- General.pou ---- *)
PROGRAM General
VAR
	WordConvertor: SafetyPLC_WordsToUDT;
	WordConvertor_v2: SafetyPLC_WordsToUDT_v2;
	test_IW132: Bools_To_Byte;
	Qtest: BYTE;
	ib26: INT;
	tbool: BOOL;
	TON_0: TON;
	TON_1: TON;
	BLINK_0: BLINK;
	restart1: BOOL;
END_VAR

%LANGUAGE LD
%NETWORK
GeneralProgramFlags(EN := TRUE);
%NETWORK
fc_Information(EN := TRUE);
%NETWORK
WordConvertor_v2(ioSafetyStatusUDT := Mach1_Safety.Status, ioSafetyControlUDT := Mach1_Safety.Control);
%NETWORK
VAR w1 : ANY; END_VAR
w1 := INVERT(HMI_Var.ForceOutputs);
Mach1_MIDS(EN := w1);
fc_Visualisation_HMI(EN := w1);
SMC_BitsToBytes(EN := w1);
%NETWORK
Status_ForceOutputs(EN := TRUE);
%NETWORK
ASSIGN(RAIL(), Q_RESET => LST_General.FirstCycle);
%NETWORK
ASSIGN(BLINK_0(ENABLE := TRUE, TIMELOW := T#1S, TIMEHIGH := T#1S), Q => Bugs.checkconnection);
%NETWORK
TON_0(IN := INVERT(Bugs.reportConnectionAlive), PT := T#2S);
%NETWORK
TON_1(IN := Bugs.reportConnectionAlive, PT := T#2S);
%NETWORK
ASSIGN(TON_0.Q OR TON_1.Q, Q => Bugs.restart);

END_PROGRAM

(* ---- Mach1_MIDS.pou ---- *)
PROGRAM Mach1_MIDS
VAR
	FB_Mach1					: GeneralMachineFlags;
	//Mach1.GenFlags				: UDT_GeneralFlags;
	tStopPositionCleaning	: BOOL;

	tDoorUnitOk				: BOOL;
	tCrossDoorcircuit1 		: BOOL;
	tCrossDoorcircuit2 		: BOOL;
	tAlarmlamp				: BOOL;
	tBool					: BOOL;
	tCond					: BOOL;

	tStopPositionLeafCarrier: BOOL;
	tReset: BOOL;
	a:INT;
//TODO
	//test5: CTD;
	//HMI_Var_Mach1_MuteNoBunchAlarm: SR;
	RepetitionNoBunch: CTD;
	tCampulseCigarPresent: BOOL;
	RepetitionNoCigar: CTD;
	PhotocellCigarHasBeenOff: SR;
	tTime1: TIME;
	tLowLevel: BOOL;
	tErrorRuntimeGreasingSystem: BOOL;
	tAlarmSL: BOOL;
	tWarningSL: BOOL;
	tStandbySL: BOOL;
	tRunningSL: BOOL;
	tHeater1Word: WORD;
	tHeater2Word: WORD;
	tHeater3Word: WORD;
	test3: BOOL;
	test4: BOOL;
	qw105: WORD;
	DRYER_SCALING_Heater1: LIN_TRAFO;

	DRYER_Scaling_Speed: LIN_TRAFO;
	lrDryer_ScaledSpeed: REAL;
	lrHeater1_ScaledPower:REAL; //% of max power of 1500

	lrHeater1_Analog: REAL;
	DRYER_SCALING_Heater2: LIN_TRAFO;
	lrHeater2_ScaledPower: REAL;
	DRYER_SCALING_Heater1_Analog: LIN_TRAFO;
	DRYER_SCALING_Heater2_Analog: LIN_TRAFO;
	lrHeater2_Analog: REAL;
	lrHeater3_ScaledPower: REAL;
	DRYER_SCALING_Heater3: LIN_TRAFO;
	lrHeater3_Analog: REAL;
	tspeed: REAL;
	TMR_ResetSafety: TON;
	tResetSafetyGuard: BOOL;
	TMR_StartupFan: TON;
	tElevatorUp: BOOL;
	tElevatorDown:BOOL;
	TMR_DelaySafetyModuleError: TON;
	Comm_OK: BOOL;
	TON_DelayAfterNetworkError: TON;
	REQ_RestartComm: BOOL;
	ReInitAllNodes: L_MC1P_ReinitAllNodes;
END_VAR
VAR
	Mach1_Drives_DB: Mach1_Drives;
	IDB_Dryer: Dryer;
	IDB_TrayFiller: TrayFiller;
END_VAR
%LANGUAGE LD
%NETWORK "DONE Network 1: Activating/deactivating MID-S/Trayfiller"
VAR w1 : ANY; w2 : ANY; END_VAR
w1 := TRUE;
w2 := w1 AND INVERT(Mach1_Safety.Status.Custom_ATF_Disabled);
ASSIGN(w2, Q => Mach1_AuxData.TrayfillerActive);
ASSIGN(w2, Q => HMI_Var.TrayfillerActive);
ASSIGN(w1 AND TRUE, Q => Mach1_AuxData.MIDS_Active);
%NETWORK "DONE Network 2: Main Block FB100 TODO"
ASSIGN(FB_Mach1(iStartResetSeparate := LST_General.AlwaysOff, iServiceButtonHasResetFunction := LST_General.AlwaysOff, iFirstCycle := LST_General.FirstCycle, iSignalPulse := LST_General.FF500ms, iAirPressureDoorsSeparate := LST_General.AlwaysOff, iEmergencyUnitOK := Mach1_AuxData.MIDS_Active AND Mach1_Safety.Status.EmergencyStopOK OR INVERT(Mach1_AuxData.MIDS_Active), iDoorUnitOK := Mach1_AuxData.MIDS_Active AND Mach1_Safety.Status.DoorsOK OR INVERT(Mach1_AuxData.MIDS_Active), iSTO_Enabled := Mach1_Safety.Status.STO_OK, iAirPressureOK := Mach1_AuxData.MIDS_Active AND LST_InputsOutputs.I100_0_AirpressureOK OR INVERT(Mach1_AuxData.MIDS_Active), iSwitchService := Mach1_Safety.Status.ServiceMode, iButtonService := Mach1_Safety.Status.Service_ButtonAB, iStart1 := LST_InputsOutputs.I100_1_Pushbutton_start_OP0a, iStop1 := Mach1_AuxData.MIDS_Active AND LST_InputsOutputs.I100_2_Pushbutton_stop_OP0a OR INVERT(Mach1_AuxData.MIDS_Active), iReset1 := LST_General.AlwaysOff, iAutoManual1 := LST_InputsOutputs.I100_3_Selector_switch_auto_manual_OP0a, iStart2 := Mach1_AuxData.TrayfillerActive AND LST_InputsOutputs.I132_1_PB_Start_OP2a, iStop2 := LST_InputsOutputs.I132_2_PB_Stop_OP2a OR INVERT(Mach1_AuxData.TrayfillerActive), iReset2 := LST_General.AlwaysOff, iAutoManual2 := LST_InputsOutputs.I132_3_SW_Auto_Man, iStart3 := LST_General.AlwaysOff, iStop3 := TRUE, iReset3 := LST_General.AlwaysOff, iAutoManual3 := LST_General.AlwaysOff, iPreDelayAfterEmergStop := T#4S, iPreStartDelayAuxDrives := OPERAND('fc_dinttotime(Mach1_Data.Timers.StartDelayAuxDrives,2)'), iPreStopDelayAuxDrives := OPERAND('fc_dinttotime(Mach1_Data.Timers.StopDelayAuxDrives,2)'), iPreDelayAfterSTOEnabled := T#2S, GenFlags := Mach1.GenFlags, oStart1 => LST_InputsOutputs.Q100_5_Signal_lamp_Start, oStop1 => LST_InputsOutputs.Q100_6_Signal_lamp_Stop, oCrossingDoorCircuit1 => tCrossDoorcircuit1, oStart2 => LST_InputsOutputs.Q132_0_SL_Start_OP2a, oStop2 => LST_InputsOutputs.Q132_1_SL_Stop_OP2a, oCrossingDoorCircuit2 => tCrossDoorcircuit2, oAlarm => tAlarmlamp), Q => tResetSafetyGuard);
%NETWORK
VAR w3 : ANY; END_VAR
w3 := TRUE;
ASSIGN(w3 AND (mach1.Genflags.StartFlag OR tResetSafetyGuard), Q_SET => Mach1_Safety.Control.ResetSafetyGuard);
ASSIGN(TMR_ResetSafety(IN := w3 AND Mach1_Safety.Control.ResetSafetyGuard, PT := T#1S), Q_RESET => Mach1_Safety.Control.ResetSafetyGuard);
%NETWORK "DONE Network 3 :Muting zones "
VAR w4 : ANY; END_VAR
w4 := TRUE AND Mach1_AuxData.MainDriveHomed AND Mach1_AuxData.RollingDeviceHomed;
ASSIGN(w4 AND tCrossDoorcircuit1, Q => Mach1_Safety.Control.Muting_zone1);
ASSIGN(w4 AND tCrossDoorcircuit1, Q => Mach1_Safety.Control.Muting_zone2);
%NETWORK "DONE NETWORK 4 (p1)Major alarms (start-up conditions)"
Alarms_V5_1_100(AlarmDB := Mach1_Alarms, iCond := Mach1_AuxData.MIDS_Active AND INVERT(Mach1_Safety.Status.EmergencyStopOK), iReset := TRUE, iAlm := Mach1_Alarms.Alm001, ioAction := Mach1.GenFlags.MajorAlarm);
%NETWORK "DONE NETWORK 4 (p2)Major alarms (start-up conditions)"
Alarms_V5_1_100(AlarmDB := Mach1_Alarms, iCond := Mach1_AuxData.MIDS_Active AND Mach1_Safety.Status.EmergencyStopOK AND (INVERT(Mach1_Safety.Status.DoorsOK) OR Mach1_Safety.Status.ServiceMode AND INVERT(Mach1_AuxData.AllDrivesHomed) AND INVERT(Mach1_Safety.Status.AllDoorsActuallyClosed)), iReset := TRUE, iAlm := Mach1_Alarms.Alm002, ioAction := Mach1.GenFlags.MinorAlarm);
%NETWORK "DONE NETWORK 4 (p3)Major alarms (start-up conditions)"
Alarms_V5_1_100(AlarmDB := Mach1_Alarms, iCond := Mach1_AuxData.MIDS_Active AND Mach1.Genflags.DelayAfterEmergStop AND INVERT(LST_InputsOutputs.I100_0_AirpressureOK), iReset := Mach1.GenFlags.StartFlag, iAlm := Mach1_Alarms.Alm004, ioAction := Mach1.GenFlags.MajorAlarm);
%NETWORK "DONE NETWORK 4 (p4)Major alarms (start-up conditions)"
ASSIGN(ASSIGN(Alarms_V5_1_100(AlarmDB := Mach1_Alarms, iCond := TMR_DelaySafetyModuleError(IN := Mach1_AuxData.MIDS_Active AND (Mach1_Safety.Status.ErrorInInputModule OR Mach1_Safety.Status.ErrorInOutputModule), PT := T#1S), iReset := TRUE, iAlm := Mach1_Alarms.Alm009, ioAction := Mach1.GenFlags.MinorAlarm), Q_SET => Mach1.Genflags.StopDriveDirect) AND (FB_Mach1.iStart1 OR FB_Mach1.iStart2 OR FB_Mach1.iStart3), Q => Mach1_Safety.Control.ExternalRequestResetSafetyModule);
%NETWORK
ASSIGN(Axis_MainDrive.xCommunicationOK AND Axis_SideCorrection.xCommunicationOK AND Axis_FeedFowardWrapper.xCommunicationOK AND Axis_OverrollingDevice.xCommunicationOK AND Axis_Bobbin.xCommunicationOK AND Axis_Fan.xCommunicationOK AND Axis_FeedForwardADS.xCommunicationOK AND Axis_FeedForwardATF.xCommunicationOK AND Axis_Elevator.xCommunicationOK, Q => Comm_OK);
%NETWORK "DONE NETWORK 4 (p3)Major alarms (start-up conditions)"
Alarms_V5_1_100(AlarmDB := Mach1_Alarms, iCond := LST_General.StartUpDelayPLC AND INVERT(Comm_OK), iReset := Mach1.GenFlags.StartFlag OR INVERT(LST_General.StartUpDelayPLC) OR Comm_OK, iAlm := Mach1_Alarms.Alm011, ioAction := Mach1.GenFlags.Warning);
%NETWORK
ASSIGN(TON_DelayAfterNetworkError(IN := Mach1_Alarms.Alm011 AND INVERT(Mach1_Alarms.Alm011), PT := T#10000S), Q => EtherCAT_Master.xRestart, Q_SET => REQ_RestartComm);
%NETWORK
ReInitAllNodes(xExecute := REQ_RestartComm, xInitCommunication := TRUE);
%NETWORK
ASSIGN(REQ_RestartComm AND Comm_OK, Q_RESET => REQ_RestartComm);
%NETWORK "TODO NETWORK 6"
ASSIGN(MainDrive(EN := TRUE) AND Mach1.GenFlags.DriveIsRunning, Q_SET => HMI_Var.Mach1.HourCounterRunning);
%NETWORK "DONE NETWORK 6: Drives"
Mach1_Drives_DB(EN := RAIL());
%NETWORK "DONE NETWORK 7: Positioned stop leaf carrier"
VAR w5 : ANY; END_VAR
w5 := TRUE;
ASSIGN(w5 AND HMI_Var.Btn_StopLeafCarrier AND (Mach1.GenFlags.RunAuto AND Mach1.GenFlags.DriveIsRunning OR Mach1_AuxData.MemStopLeafCarrier), Q => Mach1_AuxData.MemStopLeafCarrier);
ASSIGN(fc_CamC_CP_UDT(iEN := w5, iMachinePosition := HMI_Var.Mach1.Position, iResetFlag := Mach1.GenFlags.Rotflag, ioPulse := Mach1_Data.CamControls.StopPostionLeafCarrier_CP) AND Mach1_Data.CamControls.StopPostionLeafCarrier_CP.Active AND Mach1_AuxData.MemStopLeafCarrier, Q => tStopPositionLeafCarrier);
%NETWORK "DONE NETWORK 8: Alarm Positioned stop leaf carrier"
ASSIGN(Alarms_V5_1_100(AlarmDB := Mach1_Alarms, iCond := tStopPositionLeafCarrier, iReset := INVERT(Mach1_AuxData.MemStopLeafCarrier), iAlm := Mach1_Alarms.Alm054, ioAction := Mach1.GenFlags.MinorAlarm), Q_SET => Mach1.GenFlags.StopDriveDirect);
%NETWORK "DONE NETWORK 9: Positioned stop cleaning "
VAR w6 : ANY; END_VAR
w6 := TRUE;
ASSIGN(w6 AND HMI_Var.Btn_Cleaning AND (Mach1.GenFlags.RunAuto AND Mach1.GenFlags.DriveIsRunning OR Mach1_AuxData.MemStopCleaning), Q => Mach1_AuxData.MemStopCleaning);
ASSIGN(fc_CamC_CP_UDT(iEN := w6, iMachinePosition := HMI_Var.Mach1.Position, iResetFlag := Mach1.GenFlags.Rotflag, ioPulse := Mach1_Data.CamControls.StopPostionCleaning_CP) AND Mach1_AuxData.MemStopCleaning, Q => tStopPositionCleaning);
%NETWORK "DONE NETWORK 10: Alarm Positioned stop cleaning "
ASSIGN(Alarms_V5_1_100(AlarmDB := Mach1_Alarms, iCond := tStopPositionCleaning, iReset := INVERT(Mach1_AuxData.MemStopCleaning), iAlm := Mach1_Alarms.Alm037, ioAction := Mach1.GenFlags.MinorAlarm), Q_SET => Mach1.GenFlags.StopDriveDirect);
%NETWORK "DONE NETWORK 11 (p1): Level bunch magazine alarms"
Alarms_V5_1_100(EN := RAIL(), AlarmDB := Mach1_Alarms, iCond := Mach1_AuxData.IEC_TIMERS.TON_BunchLevelWarning(IN := Mach1_AuxData.MIDS_Active AND Mach1.GenFlags.DelayAfterEmergStop AND INVERT(LST_InputsOutputs.I101_4_Level_bunch_magazine) AND HMI_Var.Test_Prod AND INVERT(HMI_Var.Btn_Cleaning) AND HMI_Var.Mach1.MuteNoBunchAlarm AND Mach1_Alarms.Alm036, PT := T#5S), iReset := LST_InputsOutputs.I101_4_Level_bunch_magazine OR HMI_Var.Test_Prod OR HMI_Var.Btn_Cleaning OR HMI_Var.Mach1.MuteNoBunchAlarm OR Mach1_Alarms.Alm036, iAlm := Mach1_Alarms.Alm073, ioAction := Mach1.GenFlags.Warning);
%NETWORK "DONE NETWORK 11 (p2): Level bunch magazine alarms"
ASSIGN(Alarms_V5_1_100(AlarmDB := Mach1_Alarms, iCond := Mach1_AuxData.IEC_TIMERS.TON_BunchLevelAlarm(IN := Mach1_AuxData.MIDS_Active AND Mach1.GenFlags.DelayAfterEmergStop AND INVERT(Mach1_Alarms.Alm036) AND INVERT(LST_InputsOutputs.I101_4_Level_bunch_magazine) AND HMI_Var.Test_Prod AND INVERT(HMI_Var.Btn_Cleaning) AND INVERT(HMI_Var.Mach1.MuteNoBunchAlarm), PT := OPERAND('fc_dinttotime(Mach1_Data.Timers.BunchMagazineEmptyTime,0)')), iReset := Mach1.GenFlags.StartFlag, iAlm := Mach1_Alarms.Alm036, ioAction := Mach1.GenFlags.MinorAlarm), Q_SET => Mach1.GenFlags.StopDriveDirect);
%NETWORK "TODO NETWORK 12: SR Bunches (JL / rolling device / outfeed)"
VAR w7 : ANY; w8 : ANY; w9 : ANY; END_VAR
w7 := fc_camc_cp_udt(iEN := RAIL(), iMachinePosition := HMI_Var.Mach1.Position, iResetFlag := Mach1.GenFlags.Rotflag, ioPulse := Mach1_Data.CamControls.BunchDetection_CP);
ASSIGN(w7 AND Mach1_AuxData.ShiftRegister.SR_bunch_present_position_3_outfeed, Q_RESET => Mach1_AuxData.ShiftRegister.SR_bunch_present_position_3_outfeed);
w8 := w7 AND Mach1_AuxData.ShiftRegister.SR_bunch_present_position_2_wrapping_device;
ASSIGN(w8, Q_SET => Mach1_AuxData.ShiftRegister.SR_bunch_present_position_3_outfeed);
ASSIGN(w8, Q_RESET => Mach1_AuxData.ShiftRegister.SR_bunch_present_position_2_wrapping_device);
w9 := w7 AND Mach1_AuxData.ShiftRegister.SR_bunch_present_position_1_JL;
ASSIGN(w9, Q_SET => Mach1_AuxData.ShiftRegister.SR_bunch_present_position_2_wrapping_device);
ASSIGN(w9, Q_RESET => Mach1_AuxData.ShiftRegister.SR_bunch_present_position_1_JL);
ASSIGN(w7 AND LST_InputsOutputs.I101_1_FC_Bunch_present, Q_SET => Mach1_AuxData.ShiftRegister.SR_bunch_present_position_1_JL);
ASSIGN(w7, Q => tBool);
%NETWORK "DONE NETWORK 13: Stop bunch infeed when cleaning is activated "
ASSIGN(Mach1_AuxData.Edge.OSP_Emptying_Cleaning(CLK := HMI_Var.Btn_Cleaning), Q_RESET => HMI_Var.Btn_BunchSupply);
%NETWORK "DONE NETWORK 14: PNV Block bunch infeed"
VAR w10 : ANY; w11 : ANY; w12 : ANY; END_VAR
w10 := TRUE;
w11 := w10 AND TRUE;
w12 := fc_CamC_CP_UDT(iEN := w11, iMachinePosition := HMI_Var.Mach1.Position, iResetFlag := LST_General.AlwaysOff, ioPulse := Mach1_Data.CamControls.BlockBunchInfeed_CP) AND TRUE;
ASSIGN(w12 AND INVERT(HMI_Var.Btn_BunchSupply), Q_SET => Mach1_AuxData.BlockBunchInfeed);
ASSIGN(w12 AND HMI_Var.Btn_BunchSupply, Q_RESET => Mach1_AuxData.BlockBunchInfeed);
ASSIGN(w11 AND INVERT(Mach1.GenFlags.DelayAfterEmergStop), Q_SET => Mach1_AuxData.BlockBunchInfeed);
ASSIGN(w10 AND Mach1.GenFlags.EnablePneumEStop AND Mach1_AuxData.BlockBunchInfeed AND INVERT(Mach1_Alarms.Alm011), Q => PneumValveTerminalSMC.Pos2A);
%NETWORK "DONE NETWORK 15: Muting of alarm $"No bunch$""
ASSIGN(Mach1_AuxData.COUNTERS.RepetitionMuteNuBunch(CD := ATD_SR(iSet := Mach1_Alarms.Alm041, iReset := tBool AND (INVERT(HMI_Var.Test_Prod) OR HMI_Var.Btn_Cleaning OR Mach1_AuxData.ShiftRegister.SR_bunch_present_position_1_JL OR INVERT(HMI_Var.Btn_BunchSupply) OR Mach1_AuxData.NumberOfMutingCyclesReached), ioSR_value := hmi_var.mach1.MuteNoBunchAlarm) AND tBool AND HMI_Var.Test_Prod AND INVERT(HMI_Var.Btn_Cleaning) AND INVERT(Mach1_AuxData.ShiftRegister.SR_bunch_present_position_1_JL), LOAD := Mach1_Alarms.Alm041, PV := OPERAND('INT_TO_WORD(Mach1_Data.Counters.BunchesFillBunchFeeder.SetValue)')), Q => Mach1_AuxData.NumberOfMutingCyclesReached);
%NETWORK "DONE NETWORK 16 (p1): Alarms Bunch"
ASSIGN(Alarms_V5_1_100(AlarmDB := Mach1_Alarms, iCond := (Mach1_AuxData.COUNTERS.RepetitionNoBunch(CD := tBool AND HMI_Var.Test_Prod AND INVERT(HMI_Var.Btn_Cleaning) AND INVERT(HMI_Var.Mach1.MuteNoBunchAlarm) AND INVERT(Mach1_AuxData.ShiftRegister.SR_bunch_present_position_1_JL), LOAD := tBool AND (INVERT(HMI_Var.Test_Prod) OR HMI_Var.Btn_Cleaning OR Mach1_AuxData.ShiftRegister.SR_bunch_present_position_1_JL OR INVERT(HMI_Var.Btn_BunchSupply) OR hmi_var.mach1.MuteNoBunchAlarm) OR Mach1.GenFlags.StartFlag AND Mach1_Alarms.Alm041, PV := OPERAND('INT_TO_WORD(Mach1_Data.Counters.MaxRepetitionNoBunch.SetValue)')) AND Mach1_AuxData.AllDrivesHomed) AND INVERT(HMI_Var.Mach1.MuteNoBunchAlarm), iReset := Mach1.GenFlags.StartFlag, iAlm := Mach1_Alarms.Alm041, ioAction := Mach1.GenFlags.MinorAlarm), Q_SET => Mach1.GenFlags.StopDriveDirect);
%NETWORK "DONE NETWORK 16 (p2): Alarms Bunch"
ASSIGN(Alarms_V5_1_100(AlarmDB := Mach1_Alarms, iCond := tBool AND INVERT(Mach1_AuxData.PhotocellBunchHasBeenOff) AND HMI_Var.Btn_BunchSupply AND Mach1_AuxData.AllDrivesHomed, iReset := Mach1.GenFlags.StartFlag, iAlm := Mach1_Alarms.Alm042, ioAction := Mach1.GenFlags.MinorAlarm), Q_SET => Mach1.GenFlags.StopDriveDirect);
%NETWORK "DONE NETWORK 16 (p3): Alarms Bunch"
ATD_SR(iSet := INVERT(LST_InputsOutputs.I101_1_FC_Bunch_present), iReset := tBool, ioSR_value := Mach1_AuxData.PhotocellBunchHasBeenOff);
%NETWORK
%NETWORK "DONE NETWORK 17 (p1): Alarms: Cigar fault"
ASSIGN(Alarms_V5_1_100(AlarmDB := Mach1_Alarms, iCond := Mach1_AuxData.COUNTERS.RepetitionNoCigar(CD := ASSIGN(fc_CamC_CP_UDT(iEN := RAIL(), iMachinePosition := HMI_Var.Mach1.Position, iResetFlag := Mach1.GenFlags.Rotflag, ioPulse := Mach1_Data.CamControls.CigarDetection_CP), Q => tBool, Q => tCampulseCigarPresent) AND HMI_Var.Test_Prod AND INVERT(HMI_Var.Btn_Cleaning) AND Mach1_AuxData.ShiftRegister.SR_bunch_present_position_3_outfeed AND INVERT(LST_InputsOutputs.I101_2_Cigar_present), LOAD := tBool AND (INVERT(HMI_Var.Test_Prod) OR HMI_Var.Btn_Cleaning OR Mach1_AuxData.ShiftRegister.SR_bunch_present_position_3_outfeed AND LST_InputsOutputs.I101_2_Cigar_present) OR Mach1.GenFlags.StartFlag AND Mach1_Alarms.Alm046, PV := OPERAND('INT_TO_WORD(Mach1_Data.Counters.MaxRepetitionNoCigars.SetValue)')) AND Mach1_AuxData.AllDrivesHomed, iReset := Mach1.GenFlags.StartFlag, iAlm := Mach1_Alarms.Alm046, ioAction := Mach1.GenFlags.MinorAlarm), Q_SET => Mach1.GenFlags.StopDriveDirect);
%NETWORK "DONE NETWORK 17 (p2): Alarms: Cigar fault"
ASSIGN(Alarms_V5_1_100(AlarmDB := Mach1_Alarms, iCond := tbool AND INVERT(Mach1_AuxData.PhotocellCigarHasBeenOff) AND Mach1_AuxData.AllDrivesHomed, iReset := Mach1.GenFlags.StartFlag, iAlm := Mach1_Alarms.Alm047, ioAction := Mach1.GenFlags.MinorAlarm), Q_SET => Mach1.GenFlags.StopDriveDirect);
%NETWORK "DONE NETWORK 17 (p3): Alarms: Cigar fault"
ATD_SR(iSet := INVERT(LST_InputsOutputs.I101_2_Cigar_present), iReset := tbool, ioSR_value := Mach1_AuxData.PhotocellCigarHasBeenOff);
%NETWORK "DONE NETWORK 18: Production counter"
ASSIGN(tBool AND Mach1_AuxData.ShiftRegister.SR_bunch_present_position_3_outfeed AND LST_InputsOutputs.I101_2_Cigar_present, Q_SET => HMI_Var.Mach1.PRDCounterIncr);
%NETWORK "DONE NETWORK 19 (p1): Set cigar present in checkRegister"
VAR w13 : ANY; w14 : ANY; w15 : ANY; END_VAR
w13 := TRUE;
ASSIGN(w13 AND tCampulseCigarPresent AND LST_InputsOutputs.I101_2_Cigar_present, Q_SET => db_CheckRegister.Positie[1].Infeed.Cigar_present_infeed);
ASSIGN(w13 AND LST_InputsOutputs.I133_2_Cigar_detected_at_cross_over, Q_SET => Mach1_AuxData.MemCigarAtCrossOver);
w14 := Mach1_AuxData.Edge.OSP_DryerZeroPoint(CLK := w13 AND LST_InputsOutputs.I133_1_PROX_zero_position_transport_ADS);
w15 := w14 AND Mach1_AuxData.MemCigarAtCrossOver;
ASSIGN(w15, Q_SET => db_CheckRegister.Positie[CTE.posCigarPresentOutfeed].Outfeed.Cigar_present_outfeed);
ASSIGN(w15, Q_RESET => Mach1_AuxData.MemCigarAtCrossOver);
ASSIGN(w14, Q_RESET => Mach1_AuxData.PreviousCycleHasOutfeedError);
ASSIGN(w14 AND Mach1_AuxData.CurrentCycleHasOutfeedError, Q_SET => Mach1_AuxData.PreviousCycleHasOutfeedError);
fc_CheckRegister(EN := w14);
ASSIGN(w14, Q_RESET => Mach1_AuxData.CurrentCycleHasOutfeedError);
ASSIGN(w14 AND db_CheckRegister.CheckRegisterError, Q_SET => Mach1_AuxData.CurrentCycleHasOutfeedError);
%NETWORK "DONE NETWORK 20: Start Fan"
VAR w16 : ANY; END_VAR
w16 := Mach1.GenFlags.EnableAuxDrive AND HMI_Var.Test_Prod AND INVERT(HMI_Var.Btn_Cleaning);
ASSIGN(w16, Q => Mach1_Data.Drives.Fan.Control.StartAuto);
TMR_StartupFan(IN := w16, PT := T#5S);
%NETWORK
ASSIGN(Alarms_V5_1_100(AlarmDB := Mach1_Alarms, iCond := INVERT(HMI_Var.Btn_Cleaning) AND Mach1.GenFlags.EnableAuxDrive AND HMI_Var.Test_Prod AND INVERT(TMR_StartupFan.Q), iReset := TRUE, iAlm := Mach1_Alarms.Alm034, ioAction := mach1.Genflags.MinorAlarm), Q_SET => mach1.Genflags.StopDriveDirect);
%NETWORK "DONE NETWORK 21: Blocking glue rod"
VAR w17 : ANY; END_VAR
w17 := Mach1.GenFlags.EnablePneumEStop AND Mach1_Safety.Status.DoorsOK;
ASSIGN(w17 AND (INVERT(Mach1_AuxData.ShiftRegister.SR_bunch_present_position_2_wrapping_device) OR INVERT(HMI_Var.Test_Prod) OR HMI_Var.Btn_Cleaning) AND Mach1_AuxData.AllDrivesHomed AND INVERT(Mach1_Alarms.Alm011), Q => PneumValveTerminalSMC.Pos3A);
ASSIGN(w17 AND INVERT(PneumValveTerminalSMC.Pos3A), Q => PneumValveTerminalSMC.Pos3B);
%NETWORK "DONE NETWORK 22 (p1): Insert needle "
ASSIGN(fc_CamC_LS_UDT(iEnable := Mach1_Safety.Status.DoorsOK AND Mach1.GenFlags.EnablePneumEStop, iActualSpeed := HMI_Var.Mach1.ActualSpeed, iActualPos := HMI_Var.Mach1.Position, iRotflag := Mach1.GenFlags.Rotflag, ioUDTCamControlLS := Mach1_Data.CamControls.InserNeedle_CLS) AND Mach1_AuxData.AllDrivesHomed AND INVERT(Mach1_Alarms.Alm011), Q => PneumValveTerminalSMC.Pos4A);
%NETWORK "DONE NETWORK 22 (p2): Insert needle "
ASSIGN(Mach1_Safety.Status.DoorsOK AND Mach1.GenFlags.EnablePneumEStop AND INVERT(PneumValveTerminalSMC.Pos4A), Q => PneumValveTerminalSMC.Pos4B);
%NETWORK "DONE NETWORK 23 (p1): Bunch positioner"
ASSIGN(fc_CamC_LS_UDT(iEnable := Mach1_Safety.Status.DoorsOK AND Mach1.GenFlags.EnablePneumEStop, iActualSpeed := HMI_Var.Mach1.ActualSpeed, iActualPos := HMI_Var.Mach1.Position, iRotflag := Mach1.GenFlags.Rotflag, ioUDTCamControlLS := Mach1_Data.CamControls.BunchPositioner_CLS) AND Mach1_AuxData.AllDrivesHomed AND INVERT(Mach1_Alarms.Alm011), Q => PneumValveTerminalSMC.Pos5A);
%NETWORK "DONE NETWORK 23 (p2): Bunch positioner"
ASSIGN(Mach1_Safety.Status.DoorsOK AND Mach1.GenFlags.EnablePneumEStop AND INVERT(PneumValveTerminalSMC.Pos5A), Q => PneumValveTerminalSMC.Pos5B);
%NETWORK "DONE NETWORK 24: Manual glue pumping"
VAR w18 : ANY; w19 : ANY; END_VAR
w18 := Mach1_AuxData.EnableGlueSprayCalibration;
w19 := w18 AND TRUE AND (HMI_Var.Mach1.GlueStart OR HMI_Var.Mach1.GlueStop OR HMI_Var.Mach1.GlueReset OR HMI_Var.Mach1.SprayStart OR HMI_Var.Mach1.SprayStop OR HMI_Var.Mach1.SprayReset OR Mach1_AuxData.ScreenForOperatorSettingsActivated);
ASSIGN(w19, Q => Mach1_AuxData.ScreenForOperatorSettingsActivated);
ASSIGN(w19, Q_SET => Mach1.GenFlags.StopDriveDirect);
MOVE(EN := w18 AND (HMI_Var.Mach1.GlueReset OR INVERT(LST_InputsOutputs.I100_2_Pushbutton_stop_OP0a)), 0, OUT => Mach1_Data.Settings.Ints.ActualNumberOfGluePulses);
ASSIGN(LT(EN := w18 AND Mach1.GenFlags.EnablePneumEStop AND BRANCH_SHORTCIRCUIT((HMI_Var.Mach1.GlueStart OR LST_InputsOutputs.I100_4_Pushbutton_request_glue_OP0a) AND INVERT(LST_General.FF500ms), Mach1_AuxData.GlueWeighingCycleStarted) AND INVERT(HMI_Var.Mach1.GlueStop) AND INVERT(HMI_Var.Mach1.GlueReset) AND LST_InputsOutputs.I100_2_Pushbutton_stop_OP0a, Mach1_Data.Settings.Ints.ActualNumberOfGluePulses, Mach1_Data.Settings.Ints.MaxNumberOfGluePulses).OUT, Q => Mach1_AuxData.GlueWeighingCycleStarted);
ADD(EN := Mach1_AuxData.Edge.OSN_Gluepump(CLK := w18 AND PneumValveTerminalSMC.Pos6A) AND Mach1_AuxData.GlueWeighingCycleStarted, Mach1_Data.Settings.Ints.ActualNumberOfGluePulses, 1, OUT => Mach1_Data.Settings.Ints.ActualNumberOfGluePulses);
%NETWORK "DONE NETWORK 25: Continuous Glueing"
VAR w20 : ANY; w21 : ANY; END_VAR
w20 := TRUE;
w21 := NOT(Mach1_AuxData.Edge.OSPushbuttonGlue(CLK := w20 AND (LST_InputsOutputs.I100_4_Pushbutton_request_glue_OP0a OR Mach1_AuxData.IEC_TIMERS.TON_StopContGluePumping.Q))) AND Mach1.GenFlags.EnablePneumEStop AND INVERT(Mach1.GenFlags.DriveIsRunning) AND INVERT(Mach1_AuxData.ScreenForOperatorSettingsActivated) AND (LST_InputsOutputs.I100_4_Pushbutton_request_glue_OP0a OR Mach1_AuxData.IEC_TIMERS.DelayContiniousGluePumping.Q);
ASSIGN(w21, Q => Mach1_AuxData.MemContinuousGluePumping);
Mach1_AuxData.IEC_TIMERS.DelayContiniousGluePumping(IN := w21, PT := T#3S);
Mach1_AuxData.IEC_TIMERS.TON_StopContGluePumping(IN := w20 AND Mach1_AuxData.MemContinuousGluePumping, PT := T#120S);
%NETWORK "DONE NETWORK 26: PNV Glue pump 1+2+3"
ASSIGN(BRANCH_SHORTCIRCUIT(fc_CamC_CC_UDT(iEnable := Mach1.GenFlags.EnablePneumEStop, iMachinePosition := HMI_Var.Mach1.Position, ioCamControl := Mach1_Data.CamControls.GluePump123_C) AND Mach1_AuxData.ShiftRegister.SR_bunch_present_position_1_JL AND HMI_Var.Test_Prod AND INVERT(HMI_Var.Btn_Cleaning) AND INVERT(Mach1_AuxData.MemContinuousGluePumping) AND INVERT(Mach1_AuxData.ScreenForOperatorSettingsActivated), BRANCH_SHORTCIRCUIT(FEED := Mach1.GenFlags.EnablePneumEStop, LST_General.FF500ms AND Mach1_AuxData.MemContinuousGluePumping, LST_General.FF500ms AND Mach1_AuxData.GlueWeighingCycleStarted)) AND INVERT(Mach1_Alarms.Alm011), Q => PneumValveTerminalSMC.Pos6A, Q => LST_InputsOutputs.Q101_2_Enable_GluePump);
%NETWORK "DONE NETWORK 27: PNV Glue pump 4"
ASSIGN(BRANCH_SHORTCIRCUIT(fc_CamC_CC_UDT(iEnable := Mach1.GenFlags.EnablePneumEStop, iMachinePosition := HMI_Var.Mach1.Position, ioCamControl := Mach1_Data.CamControls.GluePump4_C) AND Mach1_AuxData.ShiftRegister.SR_bunch_present_position_1_JL AND HMI_Var.Test_Prod AND INVERT(HMI_Var.Btn_Cleaning) AND INVERT(Mach1_AuxData.MemContinuousGluePumping) AND INVERT(Mach1_AuxData.ScreenForOperatorSettingsActivated), BRANCH_SHORTCIRCUIT(FEED := Mach1.GenFlags.EnablePneumEStop, LST_General.FF500ms AND Mach1_AuxData.MemContinuousGluePumping, LST_General.FF500ms AND Mach1_AuxData.GlueWeighingCycleStarted)) AND INVERT(Mach1_Alarms.Alm011), Q => PneumValveTerminalSMC.Pos10A);
%NETWORK "DONE NETWORK 28: PNV Glue pump 5"
ASSIGN(BRANCH_SHORTCIRCUIT(fc_CamC_CC_UDT(iEnable := Mach1.GenFlags.EnablePneumEStop, iMachinePosition := HMI_Var.Mach1.Position, ioCamControl := Mach1_Data.CamControls.GluePump5_C) AND Mach1_AuxData.ShiftRegister.SR_bunch_present_position_1_JL AND HMI_Var.Test_Prod AND INVERT(HMI_Var.Btn_Cleaning) AND INVERT(Mach1_AuxData.MemContinuousGluePumping) AND INVERT(Mach1_AuxData.ScreenForOperatorSettingsActivated), BRANCH_SHORTCIRCUIT(FEED := Mach1.GenFlags.EnablePneumEStop, LST_General.FF500ms AND Mach1_AuxData.MemContinuousGluePumping, LST_General.FF500ms AND Mach1_AuxData.GlueWeighingCycleStarted)) AND INVERT(Mach1_Alarms.Alm011), Q => PneumValveTerminalSMC.Pos11A);
%NETWORK "DONE NETWORK 29: PNV Small gripper"
ASSIGN(fc_CamC_LS_UDT(iEnable := Mach1.GenFlags.EnablePneumEStop, iActualSpeed := HMI_Var.Mach1.ActualSpeed, iActualPos := HMI_Var.Mach1.Position, iRotflag := Mach1.GenFlags.Rotflag, ioUDTCamControlLS := Mach1_Data.CamControls.SmallGripper_CLS) AND Mach1_AuxData.AllDrivesHomed AND INVERT(Mach1_Alarms.Alm011), Q => PneumValveTerminalSMC.Pos7A);
%NETWORK "DONE NETWORK 30: Big gripper"
ASSIGN(fc_CamC_LS_UDT(iEnable := Mach1.GenFlags.EnablePneumEStop, iActualSpeed := HMI_Var.Mach1.ActualSpeed, iActualPos := HMI_Var.Mach1.Position, iRotflag := Mach1.GenFlags.Rotflag, ioUDTCamControlLS := Mach1_Data.CamControls.BigGripper_CLS) AND Mach1_AuxData.AllDrivesHomed AND INVERT(Mach1_Alarms.Alm011), Q => PneumValveTerminalSMC.Pos8A);
%NETWORK "TODO NETWORK 31: Blow off wrapper"
ASSIGN(fc_CamC_CC_UDT(iEnable := Mach1.GenFlags.EnablePneumEStop, iMachinePosition := HMI_Var.Mach1.Position, ioCamControl := Mach1_Data.CamControls.BlowOffWrapper_C) AND INVERT(Mach1_Alarms.Alm011), Q => PneumValveTerminalSMC.Pos9A);
%NETWORK "DONE NETWORK 32: Blow off bobbin"
ASSIGN(fc_CamC_CC_UDT(iEnable := Mach1.GenFlags.EnablePneumEStop AND Mach1.GenFlags.DriveIsRunning, iMachinePosition := HMI_Var.Mach1.Position, ioCamControl := Mach1_Data.CamControls.BlowOffBobine_C) AND INVERT(Mach1_Alarms.Alm011), Q => PneumValveTerminalSMC.Pos1A);
%NETWORK "DONE NETWORK 33: "
AHWF(EN := RAIL());
%NETWORK "TODO NETWORK 34: OBSOLETE"
%NETWORK "DONE NETWORK 35: Main FB:  Dryer-trayfiller"
VAR w22 : ANY; END_VAR
w22 := IDB_Dryer(iGenFlags := Mach1.GenFlags, iMachineStarted := Mach1.GenFlags.EnableAuxDrive AND Mach1_Safety.Status.DoorsOK AND INVERT(Mach1.GenFlags.StopFlag), iSwitchDryer := HMI_Var.Btn_DryerOn, iDryerClosed := LST_InputsOutputs.I133_0_PROX_Dryer_closed, iStartFeedForward := ASSIGN(fc_CamC_CP_UDT(iEN := RAIL(), iMachinePosition := HMI_Var.Mach1.Position, iResetFlag := Mach1.GenFlags.Rotflag, ioPulse := Mach1_Data.CamControls.FeedforwardDryer_CP), Q => Mach1_AuxData.StartpulseDryer), iStopFeedForward := (INVERT(Mach1.GenFlags.EnableAuxDrive) OR LT(EN := RAIL(), Mach1_AuxData.COUNTERS.EmptyingCycles.CV, 105).OUT OR INVERT(Trayfiller_Data.commInterface.Permission) OR INVERT(Mach1_Safety.Status.DoorsOK)) AND LST_InputsOutputs.I133_1_PROX_zero_position_transport_ADS OR Mach1_Alarms.Alm048, iPermissionDownstream := Trayfiller_Data.commInterface.Permission AND INVERT(Mach1_Alarms.Alm053), iSetPowerHeater1 := Mach1_Data.Dryer.Heater1.SetHeaterPower, iSetPowerHeater2 := Mach1_Data.Dryer.Heater2.SetHeaterPower, iSetPowerHeater3 := Mach1_Data.Dryer.Heater3.SetHeaterPower, iPowerOrAnalog := TRUE, iSpeedForEmptying := 100, oEnableHeaters => HMI_Var.Mach1.HeatersActive, oPowerHeater1 => tHeater1Word, oPowerHeater2 => tHeater2Word, oPowerHeater3 => tHeater3Word);
ASSIGN(w22 AND HMI_Var.Mach1.HeatersActive, Q => LST_InputsOutputs.Q132_2_Enable_power_controllers);
MOVE(EN := GE(EN := w22, Mach1_Data.Dryer.Heater1.SetHeaterPower, 350).OUT, 350, OUT => Mach1_Data.Dryer.Heater1.SetHeaterPower);
MOVE(EN := GE(EN := w22, Mach1_Data.Dryer.Heater2.SetHeaterPower, 350).OUT, 350, OUT => Mach1_Data.Dryer.Heater2.SetHeaterPower);
MOVE(EN := GE(EN := w22, Mach1_Data.Dryer.Heater3.SetHeaterPower, 350).OUT, 350, OUT => Mach1_Data.Dryer.Heater3.SetHeaterPower);
%NETWORK "DONE NETWORK 36: CT Fan dryer"
ASSIGN(Mach1_AuxData.TrayfillerActive AND Mach1.GenFlags.EnableAuxDrive AND HMI_Var.Btn_DryerOn, Q => LST_InputsOutputs.Q132_4_CT_Fan_dryer);
%NETWORK "TODO NETWORK 37: "
VAR w23 : ANY; END_VAR
// dryer speed: 100rpm ->1000 0.1rpm
// max AO-value: 2^14=16384
//
w23 := TRUE;
DRYER_Scaling_Speed(EN := w23, IN := OPERAND('DINT_TO_REAL(HMI_Var.Mach1.ActualSpeedDryer)'), IN_MIN := 0, IN_MAX := 1000, OUT_MIN := 0, OUT_MAX := 1, OUT => lrDryer_ScaledSpeed);
MOVE(EN := DRYER_SCALING_Heater1_Analog(EN := MOVE(EN := DRYER_SCALING_Heater1(EN := w23, IN := tHeater1Word, IN_MIN := 0, IN_MAX := 1500, OUT_MIN := 0, OUT_MAX := 1, OUT => lrHeater1_ScaledPower), OPERAND('REAL_TO_INT(lrHeater1_ScaledPower*lrDryer_ScaledSpeed*1500)'), OUT => HMI_Var.Mach1.ActHeater1), IN := OPERAND('lrDryer_ScaledSpeed*lrHeater1_ScaledPower*1500'), IN_MIN := 0, IN_MAX := 1500, OUT_MIN := 0, OUT_MAX := 16384, OUT => lrHeater1_Analog), OPERAND('REAL_TO_WORD(lrHeater1_Analog)'), OUT => %QW105);
MOVE(EN := DRYER_SCALING_Heater2_Analog(EN := MOVE(EN := DRYER_SCALING_Heater2(EN := w23, IN := tHeater2Word, IN_MIN := 0, IN_MAX := 1500, OUT_MIN := 0, OUT_MAX := 1, OUT => lrHeater2_ScaledPower), OPERAND('REAL_TO_INT(lrHeater2_ScaledPower*lrDryer_ScaledSpeed*1500)'), OUT => HMI_Var.Mach1.ActHeater2), IN := OPERAND('lrDryer_ScaledSpeed*lrHeater2_ScaledPower*1500'), IN_MIN := 0, IN_MAX := 1500, OUT_MIN := 0, OUT_MAX := 16384, OUT => lrHeater2_Analog), OPERAND('REAL_TO_WORD(lrHeater2_Analog)'), OUT => %QW106);
MOVE(EN := DRYER_SCALING_Heater2_Analog(EN := MOVE(EN := DRYER_SCALING_Heater3(EN := w23, IN := tHeater3Word, IN_MIN := 0, IN_MAX := 1500, OUT_MIN := 0, OUT_MAX := 1, OUT => lrHeater3_ScaledPower), OPERAND('REAL_TO_INT(lrHeater3_ScaledPower*lrDryer_ScaledSpeed*1500)'), OUT => HMI_Var.Mach1.ActHeater3), IN := OPERAND('lrDryer_ScaledSpeed*lrHeater3_ScaledPower*1500'), IN_MIN := 0, IN_MAX := 1500, OUT_MIN := 0, OUT_MAX := 16384, OUT => lrHeater3_Analog), OPERAND('REAL_TO_WORD(lrHeater3_Analog)'), OUT => %QW107);
%NETWORK "DONE NETWORK 38 (p1): Alarms dryer"
ASSIGN(RuntimeGuard_V5_1_100(AlarmDB := Mach1_Alarms, iForward := Mach1_AuxData.TrayfillerActive AND (IDB_Dryer.oFeedForward AND Mach1.Genflags.DelayAfterSTO OR mach1.Genflags.DriveIsRunning) AND (Mach1_AuxData.AllDrivesHomed OR INVERT(Mach1_AuxData.MIDS_Active)), iReverse := LST_General.AlwaysOff, iActivateGuard := GE(EN := Mach1.GenFlags.EnableAuxDrive AND INVERT(Mach1_Alarms.Alm048) AND (Mach1.Genflags.DelayAfterSTO AND IDB_Dryer.oFeedForward OR mach1.Genflags.DriveIsRunning) AND INVERT(LST_InputsOutputs.I133_1_PROX_zero_position_transport_ADS), Mach1_Data.Drives.FeedForwardADS.Control.AutoSpeed, 10).OUT, iMaxRuntime := T#10S, iReset := Mach1.GenFlags.StartFlag, iAlm := Mach1_Alarms.Alm048, ioAction := Mach1.GenFlags.MinorAlarm, ioAccRuntime := Mach1_AuxData.IEC_TIMERS.RuntimeGuardFeedforwardDryer, oForwardUnguarded => tBool, oForwardGuarded => Mach1_Data.Drives.FeedForwardADS.Control.StartAuto, oReverseUnguarded => tBool, oReverseGuarded => tBool), Q_SET => Mach1.GenFlags.StopDriveDirect);
%NETWORK "DONE NETWORK 38 (p2): Alarms dryer"
ASSIGN(Alarms_V5_1_100(AlarmDB := Mach1_Alarms, iCond := Mach1_AuxData.TrayfillerActive AND Mach1.GenFlags.DelayAfterEmergStop AND IDB_Dryer.oFaultDryerOpened, iReset := TRUE, iAlm := Mach1_Alarms.Alm049, ioAction := Mach1.GenFlags.MinorAlarm) AND Mach1_AuxData.AllDrivesHomed, Q_SET => Mach1.GenFlags.StopDriveDirect);
%NETWORK "TODO NETWORK 38 (p3): Alarms dryer"
VAR w24 : ANY; END_VAR
w24 := Alarms_V5_1_100(AlarmDB := Mach1_Alarms, iCond := GT(EN := mach1.Genflags.DelayAfterEmergStop AND HMI_Var.Test_Prod AND Mach1_AuxData.TrayfillerActive, Mach1_Data.Counters.MaxRepetitionNoCigarsDryer.SetValue, 0).OUT AND db_CheckRegister.CheckRegisterError AND INVERT(Mach1_AuxData.PreviousCycleHasOutfeedError), iReset := Mach1.GenFlags.StartFlag, iAlm := Mach1_Alarms.Alm053, ioAction := Mach1.GenFlags.MinorAlarm);
ASSIGN(w24, Q_SET => Mach1.GenFlags.StopDriveDirect);
ASSIGN(w24, Q_RESET => db_CheckRegister.CheckRegisterError);
%NETWORK "DONE NETWORK 38 (p4): Alarms dryer"
ASSIGN(Alarms_V5_1_100(AlarmDB := Mach1_Alarms, iCond := Mach1_AuxData.IEC_TIMERS.TON_DryerSwitchedOff(IN := Mach1_AuxData.TrayfillerActive AND HMI_Var.Test_Prod AND INVERT(HMI_Var.Btn_DryerOn), PT := T#5S), iReset := Mach1.GenFlags.StartFlag, iAlm := Mach1_Alarms.Alm058, ioAction := Mach1.GenFlags.MinorAlarm), Q_SET => Mach1.GenFlags.StopDriveDirect);
%NETWORK "TODO NETWORK 39: Analog setpoint feedforward dryer"
SpeedCalculationDryer(EN := RAIL());
%NETWORK "TODO NETWORK 40: Analog setpoint feedforward trayfiller"
SpeedCalculationTrayfiller(EN := RAIL());
%NETWORK "DONE NETWORK 41: Empty trayfiller"
ASSIGN(Mach1_AuxData.COUNTERS.EmptyingCycles(CD := HMI_Var.Btn_Cleaning AND LST_InputsOutputs.I133_1_PROX_zero_position_transport_ADS, LOAD := INVERT(HMI_Var.Btn_Cleaning), PV := 194), Q_RESET => HMI_Var.Btn_Cleaning);
%NETWORK "DONE NETWORK 42: Main block Trayfiller"
IDB_TrayFiller(iGenFlags := Mach1.GenFlags, iMachineStarted := Mach1.GenFlags.EnableAuxDrive AND INVERT(Mach1.GenFlags.StopFlag), iButtonChangeTray := LST_General.AlwaysOff, iButtonTrayDown := LST_InputsOutputs.I132_6_Tray_down, iButtonTrayUp := LST_InputsOutputs.I132_7_Tray_up, iCigarAtCrossover := LST_InputsOutputs.I133_2_Cigar_detected_at_cross_over OR LT(EN := RAIL(), Mach1_AuxData.COUNTERS.EmptyingCycles.CV, 106).OUT, iStartFeedForward := (LST_InputsOutputs.I133_1_PROX_zero_position_transport_ADS OR LT(EN := RAIL(), Mach1_AuxData.COUNTERS.EmptyingCycles.CV, 106).OUT) AND Mach1_Safety.Status.DoorsOK, iStopFeedForward := LST_InputsOutputs.I133_3_PROX_zero_position_transport_ATF, iCigarAtInpusher := LST_InputsOutputs.I133_4_Cigar_detected_at_inpusher, iRpsInpusher := LST_InputsOutputs.I133_6_PROX_inpusher_retracted, iEpsInpusher := LST_InputsOutputs.I133_7_PROX_inpusher_at_tray, iGuardInpusher := TRUE, iPsElevatorUp := LST_InputsOutputs.I136_0_PROX_Elevator_above, iPsElevatorDown := LST_InputsOutputs.I136_1_PROX_Elevator_below, iPulseCounterElevator := LST_InputsOutputs.I136_2_PROX_pulse_counter_elevator, iFcGuardTrayOnElev := LST_InputsOutputs.I136_3_FC_Position_tray_OK, iRowHeight := Mach1_Data.TrayFiller.RowHeight, iSetNumberOfRows := Mach1_Data.Trayfiller.SetNumberOfRows, iInitialDescentValue := Mach1_Data.Trayfiller.InitialDescentValue, iLightCurtainInpusher := Mach1_Safety.Status.Door_switch17, iLightCurtainElevator := Mach1_Safety.Status.Door_switch18, iPsInfeedConvAtInit := LST_InputsOutputs.I136_4_PROX_Infeed_conveyor_initial_position, iPsInfeedConvAtElev := LST_InputsOutputs.I136_5_PROX_Infeed_conveyor_at_elevator, iFcGuardTrayFromElev := LST_InputsOutputs.I136_6_FC_Guard_tray_from_elevator, iFcOutfeedConvFull := LST_InputsOutputs.I136_7_FC_Outfeed_conveyor_full, iTestProd := TRUE, ioActNumberOfRows := HMI_Var.Mach1.ActNumberOfRows, oValveTiltInpusher => LST_InputsOutputs.Q132_7_PNV_tilting_inpusher);
%NETWORK
ASSIGN(IDB_TrayFiller.oFeedForwardMotor, Q => Mach1_Data.Drives.FeedForwardATF.Control.StartAuto);
%NETWORK "DONE NETWORK 43: Selection of inpusher runtimeguard time"
VAR w25 : ANY; END_VAR
w25 := IDB_TrayFiller.oValveInpusher;
MOVE(EN := w25, T#1S, OUT => tTime1);
MOVE(EN := NOT(w25), T#5S, OUT => tTime1);
%NETWORK "DONE NETWORK 44 (p1): Runtimeguard trayfiller"
ASSIGN(RuntimeGuard_V5_1_100(AlarmDB := Mach1_Alarms, iForward := Mach1_AuxData.TrayfillerActive AND IDB_TrayFiller.oValveInpusher AND Mach1_AuxData.AllDrivesHomed, iReverse := Mach1_AuxData.TrayfillerActive AND INVERT(IDB_TrayFiller.oValveInpusher) AND Mach1_AuxData.AllDrivesHomed, iActivateGuard := Mach1_AuxData.TrayfillerActive AND Mach1.GenFlags.EnablePneumEStop AND (IDB_TrayFiller.oValveInpusher AND INVERT(LST_InputsOutputs.I133_7_PROX_inpusher_at_tray) OR INVERT(IDB_TrayFiller.oValveInpusher) AND INVERT(LST_InputsOutputs.I133_6_PROX_inpusher_retracted)), iMaxRuntime := T#3S, iReset := Mach1.GenFlags.StartFlag, iAlm := Mach1_Alarms.Alm050, ioAction := Mach1.GenFlags.MinorAlarm, ioAccRuntime := Mach1_AuxData.IEC_TIMERS.RuntimeguardInpusher, oForwardUnguarded => LST_InputsOutputs.Q132_6_PNV_Inpusher, oReverseUnguarded => tBool, oReverseGuarded => tBool), Q_SET => Mach1.GenFlags.StopDriveDirect);
%NETWORK "DONE NETWORK 44 (p2): Runtimeguard trayfiller"
ASSIGN(RuntimeGuard_V5_1_100(AlarmDB := Mach1_Alarms, iForward := Mach1_AuxData.TrayfillerActive AND IDB_TrayFiller.oElevatorMotorUp AND Mach1_AuxData.AllDrivesHomed, iReverse := Mach1_AuxData.TrayfillerActive AND IDB_TrayFiller.oElevatorMotorDown AND Mach1_AuxData.AllDrivesHomed, iActivateGuard := TRUE, iMaxRuntime := T#15S, iReset := Mach1.GenFlags.StartFlag, iAlm := Mach1_Alarms.Alm052, ioAction := Mach1.GenFlags.MinorAlarm, ioAccRuntime := Mach1_AuxData.IEC_TIMERS.RuntimeGuardElevator, oForwardGuarded => tElevatorUp, oReverseGuarded => tElevatorDown), Q_SET => Mach1.GenFlags.StopDriveDirect);
%NETWORK "DONE NETWORK 44 (p3): Runtimeguard trayfiller"
ASSIGN(RuntimeGuard_V5_1_100(AlarmDB := Mach1_Alarms, iForward := Mach1_AuxData.TrayfillerActive AND IDB_TrayFiller.oInfeedMotorFwd AND Mach1_AuxData.AllDrivesHomed, iReverse := Mach1_AuxData.TrayfillerActive AND IDB_TrayFiller.oInfeedMotorRev AND Mach1_AuxData.AllDrivesHomed, iActivateGuard := TRUE, iMaxRuntime := T#4000MS, iReset := Mach1.GenFlags.StartFlag, iAlm := Mach1_Alarms.Alm065, ioAction := Mach1.GenFlags.MinorAlarm, ioAccRuntime := Mach1_AuxData.IEC_TIMERS.RuntimeGuardInfeedConveyor, oForwardGuarded => LST_InputsOutputs.Q133_5_InfeedConv_Fwd, oReverseGuarded => LST_InputsOutputs.Q133_6_InfeedConv_Rev), Q_SET => Mach1.GenFlags.StopDriveDirect);
%NETWORK "DONE NETWORK 44 (p4): Runtimeguard trayfiller"
ASSIGN(RuntimeGuard_V5_1_100(AlarmDB := Mach1_Alarms, iForward := Mach1_AuxData.TrayfillerActive AND IDB_TrayFiller.oOutfeedMotorFwd AND Mach1_AuxData.AllDrivesHomed, iReverse := INVERT(TRUE), iActivateGuard := TRUE, iMaxRuntime := T#8500MS, iReset := Mach1.GenFlags.StartFlag, iAlm := Mach1_Alarms.Alm066, ioAction := Mach1.GenFlags.MinorAlarm, ioAccRuntime := Mach1_AuxData.IEC_TIMERS.RuntimeGuardOutfeedConveyor, oForwardUnguarded => tBool, oForwardGuarded => LST_InputsOutputs.Q133_7_OutfeedConv_Fwd, oReverseUnguarded => tBool, oReverseGuarded => tBool), Q_SET => Mach1.GenFlags.StopDriveDirect);
%NETWORK "DONE NETWORK 45: Elevator: profinet vs IO"
VAR w26 : ANY; END_VAR
w26 := tElevatorUp OR tElevatorDown;
ASSIGN(w26, Q => Mach1_Data.Drives.ElevatorATF.Control.StartAuto);
MOVE(EN := w26, 30, OUT => Mach1_Data.Drives.ElevatorATF.Control.AutoSpeed);
ASSIGN(w26 AND tElevatorDown, Q => Mach1_Data.Drives.ElevatorATF.Control.Reverse);
%NETWORK "DONE NETWORK 46 (p1): Alarms trayfiller"
ASSIGN(Alarms_V5_1_100(AlarmDB := Mach1_Alarms, iCond := Mach1_AuxData.TrayfillerActive AND Mach1.GenFlags.DelayAfterEmergStop AND Mach1.GenFlags.DelayAfterSTO AND INVERT(LST_InputsOutputs.I132_0_Thermal_guards_OK) AND (Mach1_AuxData.AllDrivesHomed OR INVERT(Mach1_AuxData.MIDS_Active)), iReset := Mach1.GenFlags.StartFlag, iAlm := Mach1_Alarms.Alm005, ioAction := Mach1.GenFlags.MinorAlarm), Q_SET => Mach1.GenFlags.StopDriveDirect);
%NETWORK "DONE NETWORK 46 (p2): Alarms trayfiller"
ASSIGN(Alarms_V5_1_100(AlarmDB := Mach1_Alarms, iCond := Mach1_AuxData.TrayfillerActive AND Trayfiller_Data.Alarms.AlmInpusherBlocked AND (Mach1_AuxData.AllDrivesHomed OR INVERT(Mach1_AuxData.MIDS_Active)), iReset := Mach1.GenFlags.StartFlag, iAlm := Mach1_Alarms.Alm059, ioAction := Mach1.GenFlags.MinorAlarm), Q_SET => Mach1.GenFlags.StopDriveDirect);
%NETWORK "DONE NETWORK 46 (p3): Alarms trayfiller"
ASSIGN(Alarms_V5_1_100(AlarmDB := Mach1_Alarms, iCond := Mach1_AuxData.TrayfillerActive AND (Trayfiller_Data.Alarms.AlmTrayPosition OR Trayfiller_Data.Alarms.AlmTrayInfeeding) AND Mach1_AuxData.AllDrivesHomed, iReset := TRUE, iAlm := Mach1_Alarms.Alm060, ioAction := Mach1.GenFlags.MinorAlarm), Q_SET => Mach1.GenFlags.StopDriveDirect);
%NETWORK "DONE NETWORK 46 (p4): Alarms trayfiller"
ASSIGN(Alarms_V5_1_100(AlarmDB := Mach1_Alarms, iCond := Mach1_AuxData.TrayfillerActive AND Trayfiller_Data.Alarms.AlmLightCurtainInpusher AND (Mach1_AuxData.AllDrivesHomed OR INVERT(Mach1_AuxData.MIDS_Active)), iReset := Mach1.GenFlags.StartFlag, iAlm := Mach1_Alarms.Alm061, ioAction := Mach1.GenFlags.MinorAlarm), Q_SET => Mach1.GenFlags.StopDriveDirect);
%NETWORK "DONE NETWORK 46 (p5): Alarms trayfiller"
Alarms_V5_1_100(AlarmDB := Mach1_Alarms, iCond := Mach1_AuxData.TrayfillerActive AND Trayfiller_Data.Alarms.WrnChangeTray AND (Mach1_AuxData.AllDrivesHomed OR INVERT(Mach1_AuxData.MIDS_Active)), iReset := TRUE, iAlm := Mach1_Alarms.Alm075, ioAction := Mach1.GenFlags.Warning);
%NETWORK "DONE NETWORK 46 (p6): Alarms trayfiller"
Alarms_V5_1_100(AlarmDB := Mach1_Alarms, iCond := Mach1_AuxData.TrayfillerActive AND Trayfiller_Data.Alarms.AlmOutfeedFull AND (Mach1_AuxData.AllDrivesHomed OR INVERT(Mach1_AuxData.MIDS_Active)), iReset := TRUE, iAlm := Mach1_Alarms.Alm062, ioAction := Mach1.GenFlags.MinorAlarm);
%NETWORK "DONE NETWORK 46 (p7): Alarms trayfiller"
Alarms_V5_1_100(AlarmDB := Mach1_Alarms, iCond := Mach1_AuxData.TrayfillerActive AND Trayfiller_Data.Alarms.AlmOutfeeding AND (Mach1_AuxData.AllDrivesHomed OR INVERT(Mach1_AuxData.MIDS_Active)), iReset := TRUE, iAlm := Mach1_Alarms.Alm063, ioAction := Mach1.GenFlags.MinorAlarm);
%NETWORK "DONE NETWORK 46 (p8): Alarms trayfiller"
ASSIGN(Alarms_V5_1_100(AlarmDB := Mach1_Alarms, iCond := Mach1_AuxData.TrayfillerActive AND Trayfiller_Data.Alarms.AlmLightCurtainElevator AND (Mach1_AuxData.AllDrivesHomed OR INVERT(Mach1_AuxData.MIDS_Active)), iReset := TRUE, iAlm := Mach1_Alarms.Alm064, ioAction := Mach1.GenFlags.MinorAlarm), Q_SET => Mach1.GenFlags.StopDriveDirect);
%NETWORK "DONE NETWORK 46 (p9): Alarms trayfiller"
ASSIGN(Mach1_AuxData.AllDrivesHomed AND Mach1_AuxData.TrayfillerActive AND INVERT(Trayfiller_Data.commInterface.Permission), Q_SET => Mach1.GenFlags.StopDriveDirect);
%NETWORK "TODO NETWORK 47 (p1):Greasing system"
%NETWORK "DONE NETWORK 47 (p2): Greasing system"
ASSIGN(Alarms_V5_1_100(AlarmDB := Mach1_Alarms, iCond := Mach1.GenFlags.DelayAfterEmergStop AND tLowLevel, iReset := TRUE, iAlm := Mach1_Alarms.Alm078, ioAction := Mach1.GenFlags.Warning), Q_SET => Mach1.GenFlags.StopDriveDirect);
%NETWORK "DONE NETWORK 48: Alarm: Greasing system"
ASSIGN(Alarms_V5_1_100(AlarmDB := Mach1_Alarms, iCond := Mach1.GenFlags.DelayAfterEmergStop AND tErrorRuntimeGreasingSystem, iReset := Mach1.GenFlags.StartFlag, iAlm := Mach1_Alarms.Alm067, ioAction := Mach1.GenFlags.MinorAlarm), Q_SET => Mach1.GenFlags.StopDriveDirect);
%NETWORK "DONE NETWORK 49: State of the machine"
VAR w27 : ANY; w28 : ANY; w29 : ANY; END_VAR
w27 := TRUE;
ASSIGN(MOVE(EN := w27 AND (Mach1.GenFlags.MajorAlarm OR Mach1.GenFlags.MinorAlarm), 0, OUT => HMI_Var.Mach1.Status), Q => tAlarmSL);
w28 := w27 AND INVERT(Mach1.GenFlags.MajorAlarm) AND INVERT(Mach1.GenFlags.MinorAlarm);
ASSIGN(MOVE(EN := w28 AND Mach1.GenFlags.Warning, 1, OUT => HMI_Var.Mach1.Status), Q => tWarningSL);
w29 := w28 AND INVERT(Mach1.GenFlags.Warning);
ASSIGN(MOVE(EN := w29 AND INVERT(Mach1.GenFlags.RunMan) AND INVERT(Mach1.GenFlags.RunAuto), 2, OUT => HMI_Var.Mach1.Status), Q => tStandbySL);
ASSIGN(MOVE(EN := w29 AND (Mach1.GenFlags.RunMan OR Mach1.GenFlags.RunAuto), 3, OUT => HMI_Var.Mach1.Status), Q => tRunningSL);
%NETWORK "TODO NETWORK 50: SL Alarmlamp"
VAR w30 : ANY; END_VAR
w30 := TRUE;
ASSIGN(w30 AND tAlarmlamp AND tAlarmSL, Q => LST_InputsOutputs.Q100_2_Pilot_light_Alarm_red_);
ASSIGN(w30 AND tAlarmlamp AND tWarningSL, Q => LST_InputsOutputs.Q100_1_Pilot_light_Alarm_orange_);
ASSIGN(BRANCH_SHORTCIRCUIT(FEED := w30, tAlarmlamp AND tStandbySL, tRunningSL), Q => LST_InputsOutputs.Q100_0_Pilot_light_Alarm_green_);
%NETWORK "TODO NETWORK 51: SL Alarmlamp Buzzer"

END_PROGRAM

(* ---- SMC_BitsToBytes.pou ---- *)
PROGRAM SMC_BitsToBytes
VAR
END_VAR

%LANGUAGE ST
LST_InputsOutputs.SMC_B0.0:= BOOL_TO_BIT( PneumValveTerminalSMC.Pos1A);
LST_InputsOutputs.SMC_B0.1:= BOOL_TO_BIT( PneumValveTerminalSMC.Pos1B);
LST_InputsOutputs.SMC_B0.2:= BOOL_TO_BIT( PneumValveTerminalSMC.Pos2A);
LST_InputsOutputs.SMC_B0.3:= BOOL_TO_BIT( PneumValveTerminalSMC.Pos2B);
LST_InputsOutputs.SMC_B0.4:= BOOL_TO_BIT( PneumValveTerminalSMC.Pos3A);
LST_InputsOutputs.SMC_B0.5:= BOOL_TO_BIT( PneumValveTerminalSMC.Pos3B);
LST_InputsOutputs.SMC_B0.6:= BOOL_TO_BIT( PneumValveTerminalSMC.Pos4A);
LST_InputsOutputs.SMC_B0.7:= BOOL_TO_BIT( PneumValveTerminalSMC.Pos4B);

LST_InputsOutputs.SMC_B1.0:= BOOL_TO_BIT( PneumValveTerminalSMC.Pos5A);
LST_InputsOutputs.SMC_B1.1:= BOOL_TO_BIT( PneumValveTerminalSMC.Pos5B);
LST_InputsOutputs.SMC_B1.2:= BOOL_TO_BIT( PneumValveTerminalSMC.Pos6A);
LST_InputsOutputs.SMC_B1.3:= BOOL_TO_BIT( PneumValveTerminalSMC.Pos6B);
LST_InputsOutputs.SMC_B1.4:= BOOL_TO_BIT( PneumValveTerminalSMC.Pos7A);
LST_InputsOutputs.SMC_B1.5:= BOOL_TO_BIT( PneumValveTerminalSMC.Pos7B);
LST_InputsOutputs.SMC_B1.6:= BOOL_TO_BIT( PneumValveTerminalSMC.Pos8A);
LST_InputsOutputs.SMC_B1.7:= BOOL_TO_BIT( PneumValveTerminalSMC.Pos8B);

LST_InputsOutputs.SMC_B2.0:= BOOL_TO_BIT( PneumValveTerminalSMC.Pos9A);
LST_InputsOutputs.SMC_B2.1:= BOOL_TO_BIT( PneumValveTerminalSMC.Pos9B);
LST_InputsOutputs.SMC_B2.2:= BOOL_TO_BIT( PneumValveTerminalSMC.Pos10A);
LST_InputsOutputs.SMC_B2.3:= BOOL_TO_BIT( PneumValveTerminalSMC.Pos10B);
LST_InputsOutputs.SMC_B2.4:= BOOL_TO_BIT( PneumValveTerminalSMC.Pos11A);
LST_InputsOutputs.SMC_B2.5:= BOOL_TO_BIT( PneumValveTerminalSMC.Pos11B);
LST_InputsOutputs.SMC_B2.6:= BOOL_TO_BIT( PneumValveTerminalSMC.Pos12A);
LST_InputsOutputs.SMC_B2.7:= BOOL_TO_BIT( PneumValveTerminalSMC.Pos12B);
(*
LST_InputsOutputs.SMC_B3.0:= BOOL_TO_BIT( PneumValveTerminalSMC.Pos13A);
LST_InputsOutputs.SMC_B3.1:= BOOL_TO_BIT( PneumValveTerminalSMC.Pos13B);
LST_InputsOutputs.SMC_B3.2:= BOOL_TO_BIT( PneumValveTerminalSMC.Pos14A);
LST_InputsOutputs.SMC_B3.3:= BOOL_TO_BIT( PneumValveTerminalSMC.Pos14B);
LST_InputsOutputs.SMC_B3.4:= BOOL_TO_BIT( PneumValveTerminalSMC.Pos15A);
LST_InputsOutputs.SMC_B3.5:= BOOL_TO_BIT( PneumValveTerminalSMC.Pos15B);
LST_InputsOutputs.SMC_B3.6:= BOOL_TO_BIT( PneumValveTerminalSMC.Pos16A);
LST_InputsOutputs.SMC_B3.7:= BOOL_TO_BIT( PneumValveTerminalSMC.Pos16B);
*)

END_PROGRAM

(* ---- SMC_BytesToBits.pou ---- *)
PROGRAM SMC_BytesToBits
VAR
END_VAR

%LANGUAGE ST
LST_InputsOutputs.SMC_B0.0:= BOOL_TO_BIT( PneumValveTerminalSMC.Pos1A);
LST_InputsOutputs.SMC_B0.1:= BOOL_TO_BIT( PneumValveTerminalSMC.Pos1B);
LST_InputsOutputs.SMC_B0.2:= BOOL_TO_BIT( PneumValveTerminalSMC.Pos2A);
LST_InputsOutputs.SMC_B0.3:= BOOL_TO_BIT( PneumValveTerminalSMC.Pos2B);
LST_InputsOutputs.SMC_B0.4:= BOOL_TO_BIT( PneumValveTerminalSMC.Pos3A);
LST_InputsOutputs.SMC_B0.5:= BOOL_TO_BIT( PneumValveTerminalSMC.Pos3B);
LST_InputsOutputs.SMC_B0.6:= BOOL_TO_BIT( PneumValveTerminalSMC.Pos4A);
LST_InputsOutputs.SMC_B0.7:= BOOL_TO_BIT( PneumValveTerminalSMC.Pos4B);

LST_InputsOutputs.SMC_B1.0:= BOOL_TO_BIT( PneumValveTerminalSMC.Pos5A);
LST_InputsOutputs.SMC_B1.1:= BOOL_TO_BIT( PneumValveTerminalSMC.Pos5A);
LST_InputsOutputs.SMC_B1.2:= BOOL_TO_BIT( PneumValveTerminalSMC.Pos6A);
LST_InputsOutputs.SMC_B1.3:= BOOL_TO_BIT( PneumValveTerminalSMC.Pos6B);
LST_InputsOutputs.SMC_B1.4:= BOOL_TO_BIT( PneumValveTerminalSMC.Pos7A);
LST_InputsOutputs.SMC_B1.5:= BOOL_TO_BIT( PneumValveTerminalSMC.Pos7B);
LST_InputsOutputs.SMC_B1.6:= BOOL_TO_BIT( PneumValveTerminalSMC.Pos8A);
LST_InputsOutputs.SMC_B1.7:= BOOL_TO_BIT( PneumValveTerminalSMC.Pos8B);

LST_InputsOutputs.SMC_B2.0:= BOOL_TO_BIT( PneumValveTerminalSMC.Pos9A);
LST_InputsOutputs.SMC_B2.1:= BOOL_TO_BIT( PneumValveTerminalSMC.Pos9B);
LST_InputsOutputs.SMC_B2.2:= BOOL_TO_BIT( PneumValveTerminalSMC.Pos10A);
LST_InputsOutputs.SMC_B2.3:= BOOL_TO_BIT( PneumValveTerminalSMC.Pos10B);
LST_InputsOutputs.SMC_B2.4:= BOOL_TO_BIT( PneumValveTerminalSMC.Pos11A);
LST_InputsOutputs.SMC_B2.5:= BOOL_TO_BIT( PneumValveTerminalSMC.Pos11B);
LST_InputsOutputs.SMC_B2.6:= BOOL_TO_BIT( PneumValveTerminalSMC.Pos12A);
LST_InputsOutputs.SMC_B2.7:= BOOL_TO_BIT( PneumValveTerminalSMC.Pos12B);
(*
SMC_B3.0:= BOOL_TO_BIT( PneumValveTerminalSMC.Pos13A);
SMC_B3.1:= BOOL_TO_BIT( PneumValveTerminalSMC.Pos13B);
SMC_B3.2:= BOOL_TO_BIT( PneumValveTerminalSMC.Pos14A);
SMC_B3.3:= BOOL_TO_BIT( PneumValveTerminalSMC.Pos14B);
SMC_B3.4:= BOOL_TO_BIT( PneumValveTerminalSMC.Pos15A);
SMC_B3.5:= BOOL_TO_BIT( PneumValveTerminalSMC.Pos15B);
SMC_B3.6:= BOOL_TO_BIT( PneumValveTerminalSMC.Pos16A);
SMC_B3.7:= BOOL_TO_BIT( PneumValveTerminalSMC.Pos16B);
*)

END_PROGRAM

(* ---- Status_ForceOutputs.pou ---- *)
PROGRAM Status_ForceOutputs
VAR
END_VAR

%LANGUAGE LD
%NETWORK
VAR w1 : ANY; END_VAR
w1 := TRUE;
MOVE(EN := w1, %IB26, OUT => LST_InputsOutputs.Serv_IB100);
MOVE(EN := w1, %IB27, OUT => LST_InputsOutputs.Serv_IB101);
%NETWORK
VAR w2 : ANY; END_VAR
w2 := TRUE;
MOVE(EN := w2, %IB370, OUT => LST_InputsOutputs.Serv_IB132);
MOVE(EN := w2, %IB371, OUT => LST_InputsOutputs.Serv_IB133);
MOVE(EN := w2, %IB372, OUT => LST_InputsOutputs.Serv_IB136);
MOVE(EN := w2, %IB373, OUT => LST_InputsOutputs.Serv_IB137);
%NETWORK
ForceOutput(EN := HMI_Var.ForceOutputs);
%NETWORK
ForceOutput_1(EN := INVERT(HMI_Var.ForceOutputs));
%NETWORK

END_PROGRAM
